	                    IF (#sx_Gapping_Rvs          // Gapping needs to be applied bit
	                        AND ((#sdi_GapHeadToHeadConfiguration_Rvs > #sdi_GapHeadToHead_Rvs    // Configured head to head bigger than the actual one
	                        OR #sdi_GapHeadToHeadConfiguration_Rvs - #idi_PEC_BoSDistance / 10 + #sdi_PECtoEndDistance_Rvs > #sdi_DownstreamGapHeadToHead_Rvs
	                        OR #sdi_GapTailToHeadConfiguration_Rvs > #sdi_Gap_Rvs     // Configured gap bigger than the actual one
	                        OR #sdi_GapTailToHeadConfiguration_Rvs - #idi_PEC_BoSDistance / 10 + #sdi_PECtoEndDistance_Rvs > #sdi_DownstreamGapTailtoHead_Rvs)
	                        AND NOT #sx_RecoveryGap_Rvs)                                                // Die back recovery gap bit not active
	                        OR (((#sdi_GapHeadToHeadConfiguration_Rvs + #i_UDT_ConveyorConfiguration.ExtraGapRecovery)   // Add recovery gap to the configured
	                        > #sdi_GapHeadToHead_Rvs                                                                                 // Actual head to head distance
	                        OR (#sdi_GapHeadToHeadConfiguration_Rvs - #idi_PEC_BoSDistance / 10 + #sdi_PECtoEndDistance_Rvs + #i_UDT_ConveyorConfiguration.ExtraGapRecovery)
	                        > #sdi_DownstreamGapHeadToHead_Rvs
	                        OR (#sdi_GapTailToHeadConfiguration_Rvs + #i_UDT_ConveyorConfiguration.ExtraGapRecovery)    // Add recovery gap to the configured
	                        > #sdi_Gap_Rvs                                                                               // Actual gap between parcels
	                        OR (#sdi_GapTailToHeadConfiguration_Rvs - #idi_PEC_BoSDistance / 10 + #sdi_PECtoEndDistance_Rvs + #i_UDT_ConveyorConfiguration.ExtraGapRecovery)
	                        > #sdi_DownstreamGapTailtoHead_Rvs)
	                        AND #sx_RecoveryGap_Rvs))                                                                                // Recovery gap bit activate
	                    THEN

	                        #sdi_GapHeadToHead_Rvs -= #iq_UDT_HandShakeUp.DownstreamDisplacement;      // Increase head to head counter with conveyor downstream displacement
	                        #sdi_Gap_Rvs -= #iq_UDT_HandShakeUp.DownstreamDisplacement;     // Increase gap counter with conveyor downstream displacement

	                    ELSE

	                        #sx_Gapping_Rvs := FALSE;                   // Set gapping bit to false

	                    END_IF;

	                    IF #sx_Gapping_Rvs                              // Gapping bit active
	                        AND NOT #iq_UDT_HandShakeUp.RTR           // Ready to receive not active
	                    THEN

	                        #sx_RecoveryGap_Rvs := TRUE;                // Recovery gap activation after die back

	                    END_IF;

	                    IF #sx_RecoveryGap_Rvs                          // Recovery gap active
	                        AND NOT #sx_Gapping_Rvs                     // Gapping bit not active
	                    THEN

	                        #sx_RecoveryGap_Rvs := FALSE;               // Recovery gap disable

	                    END_IF;

	                END_REGION
	            END_IF;
	        END_REGION

	        REGION 7.6 - Ready to send and Transfer in progress
	            IF NOT #sx_ReverseDirection
	            THEN
	                REGION 7.6.1 - Forward

	                    IF #iq_UDT_HandShake.RTR                                            // Ready to receive bit
	                        AND NOT #sx_Gapping_Fwd
	                        AND #sx_AuxHeadAtEnd_Fwd                                            // Parcel is at end of conveyor
	                        AND NOT #ix_ExternalRequestDieBack
	                    THEN

	                        #iq_UDT_HandShake.TIP := TRUE;      // Transfer in progress bit
	                        #iq_UDT_HandShake.RTS := FALSE;     // Ready to send bit
	                        #sx_AuxHeadAtEnd_Fwd := FALSE;

	                    END_IF;

	                    IF #R_TRIG_TailToBegin_Fwd.Q               // Reset TIP when the parcel leaves interlock
	                    THEN

	                        #iq_UDT_HandShake.TIP := FALSE;     // Transfer in progress bit

	                    END_IF;

	                END_REGION
	            ELSE
	                REGION 7.6.2 - Reverse

	                    IF #iq_UDT_HandShakeUp.RTR                                            // Ready to receive bit
	                        AND #iq_UDT_HandShake.RTR
	                        AND NOT #sx_Gapping_Rvs
	                        AND #sx_AuxHeadAtEnd_Rvs                                            // Parcel is at end of conveyor
	                        AND NOT #ix_ExternalRequestDieBack
	                    THEN

	                        #iq_UDT_HandShakeUp.TIP := TRUE;      // Transfer in progress bit
	                        #iq_UDT_HandShakeUp.RTS := FALSE;     // Ready to send bit
	                        #sx_AuxHeadAtEnd_Rvs := FALSE;

	                    END_IF;

	                    IF #R_TRIG_TailToBegin_Rvs.Q               // Reset TIP when the parcel leaves interlock
	                    THEN

	                        #iq_UDT_HandShakeUp.TIP := FALSE;     // Transfer in progress bit

	                    END_IF;

	                END_REGION
	            END_IF;
	        END_REGION

	        REGION 7.7 - Downstream gap

	            (* This functionality is used to maintain the gap between parcel conveyor's downstream.
	               To do this, is used the downstream displacement.  *)
	            IF NOT #sx_ReverseDirection
	            THEN
	                REGION 7.7.1 - Forward

	                    IF #R_TRIG_TailToBegin_Fwd.Q                       // When the parcel's tail reach the beginning of downstream conveyor
	                    THEN

	                        #sdi_DownstreamGapTailtoHead_Fwd := 0;                     // Reset downstream gap counter

	                    END_IF;

	                    IF #sdi_DownstreamGapTailtoHead_Fwd < #ci_OverflowLimit        // Prevent integer variable overflow
	                    THEN

	                        #sdi_DownstreamGapTailtoHead_Fwd += #iq_UDT_HandShake.DownstreamDisplacement;          // Downstream displacement gap counter

	                    END_IF;

	                END_REGION
	            ELSE
	                REGION 7.7.2 - Reverse

	                    IF #R_TRIG_TailToBegin_Rvs.Q                       // When the parcel's tail reach the beginning of downstream conveyor
	                    THEN

	                        #sdi_DownstreamGapTailtoHead_Rvs := 0;                     // Reset downstream gap counter

	                    END_IF;

	                    IF #sdi_DownstreamGapTailtoHead_Rvs < #ci_OverflowLimit        // Prevent integer variable overflow
	                    THEN

	                        #sdi_DownstreamGapTailtoHead_Rvs -= #iq_UDT_HandShakeUp.DownstreamDisplacement;          // Downstream displacement gap counter

	                    END_IF;

	                END_REGION
	            END_IF;
	        END_REGION

	        REGION 7.8 - Downstream Head to Head
	            IF NOT #sx_ReverseDirection
	            THEN
	                REGION 7.8.1 - Forward

	                    #R_TRIG_Transfering_Fwd(CLK := #iq_UDT_HandShake.TIP);

	                    IF #R_TRIG_Transfering_Fwd.Q                                                           // Transfering aux bit rising trigger
	                    THEN

	                        #sdi_DownstreamGapHeadToHead_Fwd := 0;                                              // Downstream head to head reset counter

	                    END_IF;

	                    IF #sdi_DownstreamGapHeadToHead_Fwd < #ci_OverflowLimit                                 // Prevent integer variable overflow
	                    THEN

	                        #sdi_DownstreamGapHeadToHead_Fwd += #iq_UDT_HandShake.DownstreamDisplacement;       // Downstream displacement head to head counter

	                    END_IF;

	                END_REGION
	            ELSE
	                REGION 7.8.2 - Reverse

	                    #R_TRIG_Transfering_Rvs(CLK := #iq_UDT_HandShake.TIP);

	                    IF #R_TRIG_Transfering_Rvs.Q                                                           // Transfering aux bit rising trigger
	                    THEN

	                        #sdi_DownstreamGapHeadToHead_Rvs := 0;                                              // Downstream head to head reset counter

	                    END_IF;

	                    IF #sdi_DownstreamGapHeadToHead_Rvs < #ci_OverflowLimit                                 // Prevent integer variable overflow
	                    THEN

	                        #sdi_DownstreamGapHeadToHead_Rvs -= #iq_UDT_HandShakeUp.DownstreamDisplacement;       // Downstream displacement head to head counter

	                    END_IF;

	                END_REGION
	            END_IF;
	        END_REGION

	        REGION 7.9 - Energy save

	            (* Save energy functionality is used to stop conveyor if no parcels are in the system to save energy
	               Save energy function counts displacement if the photo eye do not detects parcels. The counter is reset if:
	               - Photo eye is triggered.
	               - Reset is required from external.
	               - Ready to send is active from upstream. *)

	            // Energy save sensors filter
	            IF NOT #ix_PEC_EoS OR NOT #ix_PEC_BoS
	            THEN
	                #si_EnergySaveFilter += ABS(IN := #iq_UDT_ConveyorInterface.Displacement);
	            ELSE
	                #si_EnergySaveFilter := 0;
	            END_IF;

	            IF #i_UDT_ConveyorConfiguration.Energy                                       // Energy save functionality enable from configuration
	            THEN

	                IF #sdi_AuxEnergySave_Fwd >= #i_UDT_ConveyorConfiguration.Forward_Direction.EnergySaveLenght        // Compare energy save counter with configured lenght
	                    OR #sdi_AuxEnergySave_Rvs >= #i_UDT_ConveyorConfiguration.Reverse_Direction.EnergySaveLenght
	                THEN
	                    #sx_EnergySaveActive := TRUE;                                           // Set energy save active true
	                END_IF;

	                IF ((#si_EnergySaveFilter >= #ci_MinimumParcelLength)                                  // Photo eye detects a parcel
	                    AND NOT #sx_EnergySaveActive)                                         // Energy save active bit
	                    OR #ix_ResetEnergySave                                               // Reset energy save
	                    OR (#iq_UDT_HandShakeUp.ResetEnergySave AND NOT #sx_ReverseDirection)                               // Reset energy save externaly
	                    OR (#iq_UDT_HandShake.ResetEnergySave AND #sx_ReverseDirection)
	                    OR NOT #iq_UDT_EquipmentControl.Command.AutomaticOn                  // Automatic ON from control block
	                    OR #iq_UDT_EquipmentControl.Command.Stop                             // Stop command from control block
	                THEN
	                    #sdi_AuxEnergySave_Fwd := 0;                                        // Reset energy save counter
	                    #sdi_AuxEnergySave_Rvs := 0;                                        // Reset energy save counter
	                    #sx_EnergySaveActive := FALSE;                                      // Set energy save active to false
	                ELSE
	                    // Increament displacement counter
	                    IF NOT #sx_ReverseDirection
	                    THEN
	                        #sdi_AuxEnergySave_Fwd += #iq_UDT_ConveyorInterface.Displacement;
	                    ELSE
	                        #sdi_AuxEnergySave_Rvs -= #iq_UDT_ConveyorInterface.Displacement;
	                    END_IF;
	                END_IF;

	            ELSE
	                // If energy save functionality is disable from configuration
	                #sdi_AuxEnergySave_Fwd := 0;
	                #sdi_AuxEnergySave_Rvs := 0;// Reset energy save counter
	                #sx_EnergySaveActive := FALSE;                                      // Set energy save false
	            END_IF;
	            // Reset to downstream when not already in enery save on signal of PEC
	            // When slave conveyor pass reset esave command to master conveyor

	            IF NOT #sx_ReverseDirection
	            THEN
	                #iq_UDT_HandShake.ResetEnergySave := (NOT #ix_PEC_EoS OR #sx_AuxHeadAtEnd_Fwd OR #iq_UDT_HandShake.TIP) AND NOT #sx_EnergySaveActive
	                OR (#i_UDT_ConveyorConfiguration.Forward_Direction.Mode = 1 AND #iq_UDT_HandShakeUp.ResetEnergySave);
	            ELSE
	                #iq_UDT_HandShakeUp.ResetEnergySave := (NOT #ix_PEC_BoS OR #sx_AuxHeadAtEnd_Rvs OR #iq_UDT_HandShakeUp.TIP) AND NOT #sx_EnergySaveActive
	                OR (#i_UDT_ConveyorConfiguration.Reverse_Direction.Mode = 1 AND #iq_UDT_HandShake.ResetEnergySave);
	            END_IF;
	        END_REGION

	        REGION 7.10 - Operation modes

	            // Different modes in automatic can be configured
	            // 1 - Slave
	            // 2 - Queue
	            // 3 - Bulk flow

	            IF #sx_AutomaticActive                                          // Automatic mode active
	                AND #tx_CascadeStart                                        // Cascade startup
	            THEN

	                IF NOT #sx_ReverseDirection
	                THEN

	                    CASE #i_UDT_ConveyorConfiguration.Forward_Direction.Mode OF                   // Operation mode configured

	                        1:  // Slave

	                            // Run conveyor if ready to receive if on, and conveyor is not gapping,
	                            // and not halt request and not energy save active

	                            #iq_UDT_ConveyorInterface.RunFwd := #sx_AutomaticActive     // Automatic mode active
	                            AND #sx_Ready                                               // Ready active
	                            AND NOT #ix_ExternalRequestHold                             // Halt request is not active
	                            AND NOT #sx_EnergySaveActive                                // Energy save not active
	                            AND #iq_UDT_HandShake.RTR                               // Ready to receive active
	                            AND NOT #sx_DirectionChanged;

	                            #iq_UDT_HandShakeUp.RTR := #iq_UDT_ConveyorInterface.RunFwd;

	                        2:  // Master

	                            // With queue configuration, conveyor runs if ready to receive is true.
	                            // If ready to receive is false, conveyor runs until parcel reach the end of the conveyor.

	                            // Conveyor stops if heads parcel reache the end of the conveyor and:
	                            // - Ready to receive is false
	                            // - Or die back requested.
	                            // - Or halt requested
	                            // Conveyor also stops if gapping is active or energy save mode active.

	                            #iq_UDT_ConveyorInterface.RunFwd := #sx_AutomaticActive             // Automatic mode active
	                            AND #sx_Ready                                                       // Ready active
	                            AND NOT #sx_DirectionChanged
	                            AND NOT #sx_Gapping_Fwd                                                 // Gapping request
	                            AND NOT #sx_EnergySaveActive                                        // Energy save request
	                            AND NOT #ix_ExternalRequestHold                                     // Halt requested from external
	                            AND ((NOT #ix_ExternalRequestDieBack
	                            AND #iq_UDT_HandShake.RTR)
	                            OR (NOT #sx_AuxHeadAtEnd_Fwd
	                            AND NOT #iq_UDT_HandShake.TIP)
	                            OR (#iq_UDT_HandShake.RTR
	                            AND NOT #sx_AuxHeadAtEnd_Fwd));

	                            #iq_UDT_HandShakeUp.RTR := #iq_UDT_ConveyorInterface.RunFwd;


	                        3: //Master at bulk flow

	                            #iq_UDT_ConveyorInterface.RunFwd := #sx_AutomaticActive             // Automatic mode active
	                            AND #sx_Ready                                                       // Ready active
	                            AND NOT #sx_DirectionChanged
	                            AND NOT #sx_EnergySaveActive                                        // Energy save request
	                            AND NOT #ix_ExternalRequestHold                                     // Halt requested from external
	                            AND (
	                            (NOT #ix_ExternalRequestDieBack                                     //no die back request and the downstream is running
	                            AND #iq_UDT_HandShake.RTR)
	                            OR                                                                  //..or..
	                            (#sdi_TransitionZone = 0)                                            // no parcels at the transition zone
	                            OR                                                                  //..or..
	                            (#iq_UDT_HandShake.RTR
	                            AND NOT #ix_ExternalRequestDieBack
	                            AND NOT (#sdi_TransitionZone = 0)));                                  //downstream is running and there are

	                            //If PEC is blocked, reset tracking counter
	                            IF NOT #ix_PEC_EoS THEN
	                                #sdi_TransitionZone := #sdi_PEC_EoSDistance_Fwd / 10;
	                            END_IF;

	                            //Track parcels at the zone between EoS and conveyor end (Transition Zone)
	                            #sdi_TransitionZone := #sdi_TransitionZone - ABS(#iq_UDT_ConveyorInterface.Displacement);

	                            //If Value is negative then set to 0
	                            IF #sdi_TransitionZone < 0 THEN
	                                #sdi_TransitionZone := 0;
	                            END_IF;

	                            #iq_UDT_HandShakeUp.RTR := #iq_UDT_ConveyorInterface.RunFwd;

	                    END_CASE;

	                ELSE

	                    CASE #i_UDT_ConveyorConfiguration.Reverse_Direction.Mode OF                   // Operation mode configured

	                        1:  // Slave

	                            // Run conveyor if ready to receive if on, and conveyor is not gapping,
	                            // and not halt request and not energy save active

	                            #iq_UDT_ConveyorInterface.RunRvs := #sx_AutomaticActive     // Automatic mode active
	                            AND #sx_Ready                                               // Ready active
	                            AND NOT #ix_ExternalRequestHold                             // Halt request is not active
	                            AND NOT #sx_EnergySaveActive                                // Energy save not active
	                            AND #iq_UDT_HandShakeUp.RTR                                 // Ready to receive active
	                            AND NOT #sx_DirectionChanged;

	                            #iq_UDT_HandShake.RTR := #iq_UDT_ConveyorInterface.RunRvs;

	                        2:  // Master

	                            // With queue configuration, conveyor runs if ready to receive is true.
	                            // If ready to receive is false, conveyor runs until parcel reach the end of the conveyor.

	                            // Conveyor stops if heads parcel reache the end of the conveyor and:
	                            // - Ready to receive is false
	                            // - Or die back requested.
	                            // - Or halt requested
	                            // Conveyor also stops if gapping is active or energy save mode active.

	                            #iq_UDT_ConveyorInterface.RunRvs := #sx_AutomaticActive             // Automatic mode active
	                            AND #sx_Ready                                                       // Ready active
	                            AND NOT #sx_DirectionChanged
	                            AND NOT #sx_Gapping_Rvs                                             // Gapping request
	                            AND NOT #sx_EnergySaveActive                                        // Energy save request
	                            AND NOT #ix_ExternalRequestHold                                     // Halt requested from external
	                            AND ((NOT #ix_ExternalRequestDieBack
	                            AND #iq_UDT_HandShakeUp.RTR)
	                            OR (NOT #sx_AuxHeadAtEnd_Rvs
	                            AND NOT #iq_UDT_HandShakeUp.TIP)
	                            OR (#iq_UDT_HandShakeUp.RTR
	                            AND NOT #sx_AuxHeadAtEnd_Rvs));

	                            #iq_UDT_HandShake.RTR := #iq_UDT_ConveyorInterface.RunRvs;


	                        3: //Master at bulk flow

	                            #iq_UDT_ConveyorInterface.RunRvs := #sx_AutomaticActive             // Automatic mode active
	                            AND #sx_Ready                                                       // Ready active
	                            AND NOT #sx_DirectionChanged
	                            AND NOT #sx_EnergySaveActive                                        // Energy save request
	                            AND NOT #ix_ExternalRequestHold                                     // Halt requested from external
	                            AND (
	                            (NOT #ix_ExternalRequestDieBack                                     //no die back request and the downstream is running
	                            AND #iq_UDT_HandShakeUp.RTR)
	                            OR                                                                  //..or..
	                            (#sdi_TransitionZone = 0)                                            // no parcels at the transition zone
	                            OR                                                                  //..or..
	                            (#iq_UDT_HandShakeUp.RTR
	                            AND NOT #ix_ExternalRequestDieBack
	                            AND NOT (#sdi_TransitionZone = 0)));                                  //downstream is running and there are

	                            //If PEC is blocked, reset tracking counter
	                            IF NOT #ix_PEC_BoS THEN
	                                #sdi_TransitionZone := #sdi_PEC_EoSDistance_Rvs / 10;
	                            END_IF;
	                            //Track parcels at the zone between EoS and conveyor end (Transition Zone)
	                            #sdi_TransitionZone := #sdi_TransitionZone - ABS(#iq_UDT_ConveyorInterface.Displacement);

	                            //If Value is negative then set to 0
	                            IF #sdi_TransitionZone < 0 THEN
	                                #sdi_TransitionZone := 0;
	                            END_IF;

	                            #iq_UDT_HandShake.RTR := #iq_UDT_ConveyorInterface.RunRvs;
	                    END_CASE;

	                END_IF;

	            ELSE

	                // If conveyor is not in manual mode and not ready
	                IF NOT #sx_ReverseDirection
	                THEN
	                    #iq_UDT_ConveyorInterface.RunFwd := FALSE;                      // Order to VFD stop conveyor
	                    #iq_UDT_HandShakeUp.RTR := FALSE;                               // Set ready to receive false
	                ELSE
	                    #iq_UDT_ConveyorInterface.RunRvs := FALSE;                      // Order to VFD stop conveyor
	                    #iq_UDT_HandShake.RTR := FALSE;                               // Set ready to receive false
	                END_IF;

	            END_IF;

	        END_REGION

	    END_IF;
	END_REGION

	REGION 8 - Speed control

	    (*In manual mode, conveyor default runs with manual speed which is calculated as a percentage of nominal speed. If "ManualFullSpeed" is set true, conveyor runs with high speed in manual mode.
	     In jog mode conveyor always runs in low speed. In automatic mode, conveyor runs with full speed if external is zero. If external speed is bigger than zero, conveyor will run with that speed. *)


	    // security
	    IF #iq_UDT_ConveyorCommand.ManualSpeed > 100 THEN
	        #iq_UDT_ConveyorCommand.ManualSpeed := 100;
	    END_IF;

	    IF #iq_UDT_ConveyorCommand.ManualSpeed < 0 THEN
	        #iq_UDT_ConveyorCommand.ManualSpeed := 0;
	    END_IF;



	    IF #sx_ManualModeActive                                                                         // Manual mode active
	    THEN

	        IF #iq_UDT_ConveyorCommand.ManualStartStop                                              // Full speed in manual mode
	        THEN

	            IF #iq_UDT_ConveyorCommand.ManualFullSpeed                                                  // Full speed in manual mode
	            THEN
	                #iq_UDT_ConveyorInterface.SpeedSetpoint := #i_UDT_ConveyorConfiguration.SpeedSetpointNominal;    // Move nominal setpoint to the VDF

	            ELSE
	                #iq_UDT_ConveyorInterface.SpeedSetpoint := REAL_TO_INT(INT_TO_REAL(#iq_UDT_ConveyorCommand.ManualSpeed) * (INT_TO_REAL(#i_UDT_ConveyorConfiguration.SpeedSetpointNominal) / 100));     // Calculate and Move manual speed setpoint to VFD

	            END_IF;

	        ELSE                                                                                             //low speed for jog mode

	            IF #i_UDT_ConveyorConfiguration.SpeedSetpointLow < #i_UDT_ConveyorConfiguration.SpeedSetpointNominal  //Low speed can't be higher than nominal speed
	            THEN
	                #iq_UDT_ConveyorInterface.SpeedSetpoint := #i_UDT_ConveyorConfiguration.SpeedSetpointLow;    // Move low speed setpoint to the VDF

	            ELSE

	                #iq_UDT_ConveyorInterface.SpeedSetpoint := #i_UDT_ConveyorConfiguration.SpeedSetpointNominal;    // Move low speed setpoint to the VDF
	            END_IF;
	        END_IF;



	    ELSE

	        IF #ii_ExternalSpeed > 0                                                                      // If external speed bigger than zero
	        THEN
	            #iq_UDT_ConveyorInterface.SpeedSetpoint := #ii_ExternalSpeed;                                     // Move external speed to VFD
	        ELSE
	            #iq_UDT_ConveyorInterface.SpeedSetpoint := #i_UDT_ConveyorConfiguration.SpeedSetpointNominal;       // Move nominal setpoint to VFD
	        END_IF;

	    END_IF;



	END_REGION


	REGION 9 - Status
	    #s_UDT_HMIStatus.Specific.Reverse := #sx_ReverseDirection;

	    // stopped
	    #s_UDT_CommonStatus.Stopped := NOT #sx_Ready OR NOT #sx_AutomaticActive;

	    // Auto ON
	    #s_UDT_CommonStatus.AutoON := #sx_Ready AND #sx_AutomaticActive;

	    // Running
	    #s_UDT_CommonStatus.Running := #iq_UDT_ConveyorInterface.RunFwd
	    OR #iq_UDT_ConveyorInterface.RunRvs;

	    // Halted
	    #s_UDT_CommonStatus.Halted := #ix_ExternalRequestHold
	    AND #s_UDT_CommonStatus.AutoON
	    AND NOT #s_UDT_CommonStatus.EnergySave;

	    // Energy save active
	    #s_UDT_CommonStatus.EnergySave := #sx_EnergySaveActive AND #sx_AutomaticActive;

	    // Die back
	    #s_UDT_CommonStatus.Dieback := #s_UDT_CommonStatus.AutoON
	    AND NOT #s_UDT_CommonStatus.EnergySave
	    AND NOT #s_UDT_CommonStatus.Running;

	    // Manual
	    #s_UDT_CommonStatus.Manual := #sx_ManualModeActive;

	    // Manual Running
	    #s_UDT_CommonStatus.ManualRun := #sx_ManualModeActive AND #s_UDT_CommonStatus.Running;

	    // Safety not ok
	    #s_UDT_CommonStatus.SafetyStop := NOT #ix_SafetyOk AND #ix_HardwareOk;

	    // HMI status update
	    IF #s_UDT_CommonStatusOld <> #s_UDT_CommonStatus                                            // update on change
	        OR (#R_TRIG_Reverse.Q OR #F_TRIG_Reverse.Q)
	    THEN
	        // HMI status initialization
	        #s_UDT_HMIStatus.Status := 0;


	        // Energy save
	        IF #s_UDT_CommonStatus.EnergySave
	        THEN
	            #s_UDT_HMIStatus.Status := "DB_HMIStatusConfiguration".EnergySave;
	        END_IF;

	        // Running
	        IF #s_UDT_CommonStatus.Running
	        THEN
	            #s_UDT_HMIStatus.Status := "DB_HMIStatusConfiguration".Running;
	        END_IF;

	        // Stopped
	        IF #s_UDT_CommonStatus.Stopped
	        THEN
	            #s_UDT_HMIStatus.Status := "DB_HMIStatusConfiguration".Stopped;
	        END_IF;

	        // Dieback
	        IF #s_UDT_CommonStatus.Dieback
	        THEN
	            #s_UDT_HMIStatus.Status := "DB_HMIStatusConfiguration".Dieback;
	        END_IF;

	        // Halted
	        IF #s_UDT_CommonStatus.Halted
	        THEN
	            #s_UDT_HMIStatus.Status := "DB_HMIStatusConfiguration".Halted;
	        END_IF;

	        // Manual
	        IF #s_UDT_CommonStatus.Manual
	        THEN
	            #s_UDT_HMIStatus.Status := "DB_HMIStatusConfiguration".Manual;
	        END_IF;

	        // Running in manual mode
	        IF #s_UDT_CommonStatus.ManualRun
	        THEN
	            #s_UDT_HMIStatus.Status := "DB_HMIStatusConfiguration".ManualRun;
	        END_IF;

	(*        // Internal tracking warning
	        IF #iq_UDT_ConveyorInterface.InternalWarningTracking
	        THEN
	            #s_UDT_HMIStatus.Status := "DB_HMIStatusConfiguration".Warning;
	        END_IF; *)

	        // Internal tracking error
	        IF #iq_UDT_ConveyorInterface.InternalErrorTracking
	        THEN
	            #s_UDT_HMIStatus.Status := "DB_HMIStatusConfiguration".TrackingError;
	        END_IF;

	        // Internal PEC error
	        IF #iq_UDT_ConveyorInterface.InternalErrorPEC
	        THEN
	            #s_UDT_HMIStatus.Status := "DB_HMIStatusConfiguration".PECJam;
	        END_IF;

	        // Internal Encoder error
	        IF #iq_UDT_ConveyorInterface.InternalErrorEncoder
	        THEN
	            #s_UDT_HMIStatus.Status := "DB_HMIStatusConfiguration".EncoderError;
	        END_IF;

	        // Internal VFD error
	        IF #iq_UDT_ConveyorInterface.InternalErrorVFD
	        THEN
	            #s_UDT_HMIStatus.Status := "DB_HMIStatusConfiguration".VFDError;
	        END_IF;

	        // Disconnect error
	        IF #iq_UDT_ConveyorInterface.Disconnected
	        THEN
	            #s_UDT_HMIStatus.Status := "DB_HMIStatusConfiguration".CBError;
	        END_IF;

	        // Safety stop
	        IF (#s_UDT_CommonStatus.SafetyStop)
	        THEN
	            #s_UDT_HMIStatus.Status := "DB_HMIStatusConfiguration".SafetyStop;
	        END_IF;

	        #s_UDT_CommonStatusOld := #s_UDT_CommonStatus;              // Copy status to memory
	        #q_UDT_Status := #s_UDT_CommonStatus;                       // Copy status to output

	    END_IF;

	    // Copy HMI status to output
	    #q_UDT_HMIStatus := #s_UDT_HMIStatus;

	END_REGION


	REGION 10 - Statistics

	    REGION 10.1 - Conveyor up time

	        IF #sx_Up OR #iq_UDT_EquipmentControl.Command.ResetData    // Reset statistics
	        THEN

	            "FC_Statistics"(ix_Reset := #iq_UDT_EquipmentControl.Command.ResetData,      // Reset statistics input
	                            ix_Activate := #sx_Up,
	                            ix_RTrigActivate := #R_TRIG_ConveyorUp.Q,                     // Statistics active trigger
	                            iqUDT_Statistics := #iq_UDT_Statistics.ConveyorUp);      // Statistics values output

	        END_IF;

	    END_REGION

	    REGION 10.2 - Energy save

	        // Statistics Energy save mode active
	        IF #s_UDT_CommonStatus.EnergySave(* #sx_EnergySaveActive *)                                                        // Energy save active
	            OR #iq_UDT_EquipmentControl.Command.ResetData                               // Reset statistics
	        THEN
	            "FC_Statistics"(ix_Reset := #iq_UDT_EquipmentControl.Command.ResetData,      // Reset statistics input
	                            ix_Activate := #s_UDT_CommonStatus.EnergySave,                         // Activate statistics functions input
	                            ix_RTrigActivate := #R_TRIG_EnergySave.Q,                    // Statistics active trigger
	                            iqUDT_Statistics := #iq_UDT_Statistics.EnergySave);         // Statistics values output

	        END_IF;

	    END_REGION

	    REGION 10.3 - Conveyor down time

	        // Conveyor down is when conveyor is not in manual mode and has an error
	        IF #sx_Down OR #iq_UDT_EquipmentControl.Command.ResetData OR #s_UDT_CommonStatus.SafetyStop                                    // Reset statistics
	        THEN

	            "FC_Statistics"(ix_Reset := #iq_UDT_EquipmentControl.Command.ResetData,             // Reset statistics input
	                            ix_Activate := #sx_Down OR #s_UDT_CommonStatus.SafetyStop, // Activate statistics functions input
	                            ix_RTrigActivate := #R_TRIG_ConveyorDownTime.Q,                     // Statistics active trigger
	                            iqUDT_Statistics := #iq_UDT_Statistics.ConveyorDown);              // Statistics values output

	        END_IF;
	    END_REGION

	    REGION 10.4 - Conveyor stop time

	        IF #sx_Stopped OR #iq_UDT_EquipmentControl.Command.ResetData                                           // Reset statistics
	        THEN

	            "FC_Statistics"(ix_Reset := #iq_UDT_EquipmentControl.Command.ResetData,        // Reset statistics input
	                            ix_Activate := #sx_Stopped,                                           // Activate statistics functions input
	                            ix_RTrigActivate := #R_TRIG_ConveyorStopped.Q,                        // Statistics active trigger
	                            iqUDT_Statistics := #iq_UDT_Statistics.ConveyorStop);                  // Statistics values output

	        END_IF;
	    END_REGION

	END_REGION

	REGION 11 - Report to control block
	    // Function to manage report between control block and conveyor block
	    "FC_EquipmentReport"(iUDT_Status := #s_UDT_CommonStatus,
	                         iqUDT_Control := #iq_UDT_EquipmentControl);

	END_REGION

	REGION 12 - Internal errors and warnings reset

	    IF #iq_UDT_EquipmentControl.Command.Reset
	    THEN

	        #iq_UDT_ConveyorInterface.InternalErrorEncoder := FALSE;
	        #iq_UDT_ConveyorInterface.InternalErrorPEC := FALSE;
	        #iq_UDT_ConveyorInterface.InternalWarningTracking := FALSE;
	        #iq_UDT_ConveyorInterface.InternalErrorTracking := FALSE;
	        #iq_UDT_ConveyorInterface.InternalWarningVFD := FALSE;
	        #iq_UDT_ConveyorInterface.InternalErrorVFD := FALSE;
	        #iq_UDT_ConveyorInterface.Disconnected := FALSE;
	        #iq_UDT_ConveyorInterface.ConfigurationError := FALSE;
	    END_IF;

	END_REGION






END_FUNCTION_BLOCK

FUNCTION_BLOCK "FB_ConnectionCheck1Hz"
{ S7_Optimized_Access := 'TRUE' }
VERSION : 3.2
// ATTRIBUTES
// AUTO_NUMBER = True
// BLOCK_NUMBER = 93
// END_ATTRIBUTES
   VAR_INPUT
      ix_LifebitIn { ExternalAccessible := 'False'; ExternalVisible := 'False'; ExternalWritable := 'False'} : Bool;   // Input life bit
      ix_IOModuleOK { ExternalAccessible := 'False'; ExternalVisible := 'False'; ExternalWritable := 'False'} : Bool;   // TRUE when IO module is Ok
   END_VAR

   VAR_OUTPUT
      qx_LifebitOut { ExternalAccessible := 'False'; ExternalVisible := 'False'; ExternalWritable := 'False'} : Bool;   // Generated life bit 1 sec ON/1 sec OFF
   END_VAR

   VAR_IN_OUT
      iqudt_ConnectionStatus : "UDT_ConnectStatus";   // Connection status
   END_VAR

   VAR
      FB_Pulse_Instance { ExternalAccessible := 'False'; ExternalVisible := 'False'; ExternalWritable := 'False'; S7_SetPoint := 'False'} : "FB_Pulse";
      F_TRIG_LifebitIn {InstructionName := 'F_TRIG'; LibVersion := '1.0'; ExternalAccessible := 'False'; ExternalVisible := 'False'; ExternalWritable := 'False'; S7_SetPoint := 'False'} : F_TRIG;   // Falling edge trigger Lifebit in
      R_TRIG_LifebitIn {InstructionName := 'R_TRIG'; LibVersion := '1.0'; ExternalAccessible := 'False'; ExternalVisible := 'False'; ExternalWritable := 'False'; S7_SetPoint := 'False'} : R_TRIG;   // Rising edge trigger  Lifebit in
      sx_LifebitValue { ExternalAccessible := 'False'; ExternalVisible := 'False'; ExternalWritable := 'False'} : Bool;   // Lifebit value
      sx_ConnectionFault { ExternalAccessible := 'False'; ExternalVisible := 'False'; ExternalWritable := 'False'} : Bool;   // Connection Fault
   END_VAR

   VAR_TEMP
      tx_Pulse : Bool;   // Generated pulse signal
   END_VAR

   VAR CONSTANT
      cudi_ConnectionFaultOnDelay : UDInt := 5000;   // Connection On Delay
   END_VAR


BEGIN
	(*
	----------------------------------------------------------------------------------------
	|                                                                                      |
	|  Copyright  2023             FORTNA Europe BV                                        |
	|  All Rights Reserved         Netherlands                                             |
	|                                                                                      |
	----------------------------------------------------------------------------------------

	Version history:
	Date        | Version   | Author        | Remark
	----------------------------------------------------------------------------------------
	12/10/2023  | 1.0       | S. Nikodem    | First release TIA 17 | DHL Munich
	12/03/2024  | 1.1       | S. Nieswiec      | Added to new Baseline
	*)

	REGION 1 - Life bit generations

	    //Generation
	    #qx_LifebitOut := "DB_Memory".Clock_1Hz;

	END_REGION

	REGION 2 - Hardware Ok

	    IF NOT #ix_IOModuleOK THEN

	        //Status update
	        #iqudt_ConnectionStatus.Specific.CommunicationFault := False;
	        #iqudt_ConnectionStatus.Specific.Connected := False;

	        #iqudt_ConnectionStatus.Status := 0;

	        RETURN;

	    END_IF;

	END_REGION

	REGION 3 - Connection check

	    //Trigger
	    #F_TRIG_LifebitIn(CLK := #ix_LifebitIn);
	    #R_TRIG_LifebitIn(CLK := #ix_LifebitIn);

	    IF (#F_TRIG_LifebitIn.Q OR #R_TRIG_LifebitIn.Q) THEN

	        #sx_LifebitValue := TRUE;
	    END_IF;

	    #FB_Pulse_Instance(iudi_PulseTime := #cudi_ConnectionFaultOnDelay,
	                       qx_Pulse => #tx_Pulse);

	    IF #tx_Pulse THEN
	        IF #sx_LifebitValue THEN

	            #sx_LifebitValue := False;

	            #sx_ConnectionFault := False;

	        ELSE

	            #sx_ConnectionFault := TRUE;

	        END_IF;
	    END_IF;

	END_REGION

	REGION 4 - Status update

	    #iqudt_ConnectionStatus.Specific.CommunicationFault := #sx_ConnectionFault;
	    #iqudt_ConnectionStatus.Specific.Connected := NOT #sx_ConnectionFault;

	    IF #sx_ConnectionFault
	    THEN
	        #iqudt_ConnectionStatus.Status := "DB_HMIStatusConfiguration".CommunicationError;
	    END_IF;

	    IF NOT #sx_ConnectionFault
	    THEN
	        #iqudt_ConnectionStatus.Status := "DB_HMIStatusConfiguration".AutoON;
	    END_IF;

	END_REGION
END_FUNCTION_BLOCK

FUNCTION_BLOCK "FB_Xray_Rapiscan"
{ S7_Optimized_Access := 'TRUE' }
VERSION : 0.1
// ATTRIBUTES
// AUTO_NUMBER = True
// BLOCK_NUMBER = 110
// END_ATTRIBUTES
   VAR_INPUT
      i_UDT_XrayConfiguration { ExternalAccessible := 'False'; ExternalVisible := 'False'; ExternalWritable := 'False'} : "UDT_XrayRapiscanConfiguration";   // Xray configuration structure
      ix_XrayEnergised { ExternalAccessible := 'False'; ExternalVisible := 'False'; ExternalWritable := 'False'} : Bool;   // Xray input signal - Energised
      ix_XrayFault { ExternalAccessible := 'False'; ExternalVisible := 'False'; ExternalWritable := 'False'} : Bool;   // Xray input signal - Fault
      ix_XrayReadyReceive { ExternalAccessible := 'False'; ExternalVisible := 'False'; ExternalWritable := 'False'} : Bool;   // Xray input signal - Ready receive
      ix_XrayReadySend { ExternalAccessible := 'False'; ExternalVisible := 'False'; ExternalWritable := 'False'} : Bool;   // Xray input signal - Ready send
      ix_XrayConveyorRunFwd { ExternalAccessible := 'False'; ExternalVisible := 'False'; ExternalWritable := 'False'} : Bool;   // Xray input signal - Conveyor run Fwd
      ix_XrayConveyorRunRvs { ExternalAccessible := 'False'; ExternalVisible := 'False'; ExternalWritable := 'False'} : Bool;   // Xray input signal - Conveyor run Rvs
      ix_XrayBagScaning { ExternalAccessible := 'False'; ExternalVisible := 'False'; ExternalWritable := 'False'} : Bool;   // Xray input signal - Xray bag scaning
      ix_XrayEmergencyStop { ExternalAccessible := 'False'; ExternalVisible := 'False'; ExternalWritable := 'False'} : Bool;   // Xray input signal - Emergency Stop
      ix_SafetyOk { ExternalAccessible := 'False'; ExternalVisible := 'False'; ExternalWritable := 'False'} : Bool;   // TRUE when Safety Circuit is healthy
      ix_24vOk { ExternalAccessible := 'False'; ExternalVisible := 'False'; ExternalWritable := 'False'} : Bool;   // TRUE when 24VDC is healthy
      ix_400vOk { ExternalAccessible := 'False'; ExternalVisible := 'False'; ExternalWritable := 'False'} : Bool;   // TRUE when 400VAC is healthy
      ix_HardwareOk { ExternalAccessible := 'False'; ExternalVisible := 'False'; ExternalWritable := 'False'} : Bool;   // TRUE when  hardware is Ok
      ix_SafetyReset { ExternalAccessible := 'False'; ExternalVisible := 'False'; ExternalWritable := 'False'} : Bool;   // TRUE Safety reset command is active
      is_ActualTime { ExternalAccessible := 'False'; ExternalVisible := 'False'; ExternalWritable := 'False'} : String;   // Actual date and time in String
   END_VAR

   VAR_OUTPUT
      q_UDT_HMIStatus { ExternalAccessible := 'False'; ExternalVisible := 'False'; ExternalWritable := 'False'} : "UDT_RapiscanStatus";   // HMI status structure
      qx_BHS_RDY_SEND { ExternalAccessible := 'False'; ExternalVisible := 'False'; ExternalWritable := 'False'} : Bool;   // Xray output signal - Input conveyor is ready to pass a bag to the Xray
      qx_BHS_RDY_RCV { ExternalAccessible := 'False'; ExternalVisible := 'False'; ExternalWritable := 'False'} : Bool;   // Xray output signal - Output conveyor is ready to accept a bag from the Xray
      qx_DECISION_ACK { ExternalAccessible := 'False'; ExternalVisible := 'False'; ExternalWritable := 'False'} : Bool;   // Xray output signal - Decision confirmation (only for Xray local control)
      qx_TRANSPORT_ENABLE { ExternalAccessible := 'False'; ExternalVisible := 'False'; ExternalWritable := 'False'} : Bool;   // Xray output signal - Transport mode eneble
      qx_TRANSPORT_FWD { ExternalAccessible := 'False'; ExternalVisible := 'False'; ExternalWritable := 'False'} : Bool;   // Xray output signal - Run forward request
      qx_TRANSPORT_REV { ExternalAccessible := 'False'; ExternalVisible := 'False'; ExternalWritable := 'False'} : Bool;   // Xray output signal - Run reverse request
      qx_ESTOP_IN { ExternalAccessible := 'False'; ExternalVisible := 'False'; ExternalWritable := 'False'} : Bool;   // Xray output signal - Estop
      qx_EMERGENCY_STOP_RESET { ExternalAccessible := 'False'; ExternalVisible := 'False'; ExternalWritable := 'False'} : Bool;   // Xray output signal - Estop resert
   END_VAR

   VAR_IN_OUT
      iq_UDT_Statistics : "UDT_RapiscanStatistics";   // Statistics structure
      iq_UDT_EquipmentControl : "UDT_EquipmentControl";   // Equipment control stucture
      iq_UDT_XrayConveyorInterface : "UDT_ConveyorInterface";   // Xray conveyor interface structure
      iq_UDT_Handshake : "UDT_ConveyorHandshake";   // Downstream handshake structure
      iq_UDT_HandShakeUp : "UDT_ConveyorHandshake";   // Upstream handshake structure
      iq_UDT_MFCCommand : "UDT_XrayCommand";   // Xray command structure
      iqs_XrayConveyorTrackingData : Array[*] of Int;   // Xray conveyor tracking array
      iq_UDT_XrayInterface : "UDT_XrayInterface";   // Xray interface structure
   END_VAR

   VAR
      s_EstopReset { ExternalAccessible := 'False'; ExternalVisible := 'False'; ExternalWritable := 'False'; S7_SetPoint := 'False'} : "FB_TimerOnOffDelay";   // Estop reset puls
      s_BagScaningTime { ExternalAccessible := 'False'; ExternalVisible := 'False'; ExternalWritable := 'False'; S7_SetPoint := 'False'} : "FB_TimerOnOffDelay";   // Bag scaning time
      s_UDT_HMIStatus { ExternalAccessible := 'False'; ExternalVisible := 'False'; ExternalWritable := 'False'; S7_SetPoint := 'False'} : "UDT_RapiscanStatus";   // HMI status structure
      s_UDT_CommonStatusOld { ExternalAccessible := 'False'; ExternalVisible := 'False'; ExternalWritable := 'False'; S7_SetPoint := 'False'} : "UDT_CommonStatus";   // Common status structure
      s_UDT_CommonStatus { ExternalAccessible := 'False'; ExternalVisible := 'False'; ExternalWritable := 'False'; S7_SetPoint := 'False'} : "UDT_CommonStatus";   // Common status structure
      R_TRIG_TransportMode {InstructionName := 'R_TRIG'; LibVersion := '1.0'; ExternalAccessible := 'False'; ExternalVisible := 'False'; ExternalWritable := 'False'; S7_SetPoint := 'False'} : R_TRIG;   // Rising edge trigger of Xray transport mode signal
      R_TRIG_XrayBagScaning {InstructionName := 'R_TRIG'; LibVersion := '1.0'; ExternalAccessible := 'False'; ExternalVisible := 'False'; ExternalWritable := 'False'; S7_SetPoint := 'False'} : R_TRIG;   // Rising edge trigger of Xray b ag scaning signal
      F_TRIG_XrayBagScaning {InstructionName := 'F_TRIG'; LibVersion := '1.0'; ExternalAccessible := 'False'; ExternalVisible := 'False'; ExternalWritable := 'False'; S7_SetPoint := 'False'} : F_TRIG;   // Falling edge trigger of Xray b ag scaning signal
      R_TRIG_SystemReadyRcv {InstructionName := 'R_TRIG'; LibVersion := '1.0'; ExternalAccessible := 'False'; ExternalVisible := 'False'; ExternalWritable := 'False'; S7_SetPoint := 'False'} : R_TRIG;   // Rising edge trigger of System ready to receive signal
      F_TRIG_SystemReadyRcv {InstructionName := 'F_TRIG'; LibVersion := '1.0'; ExternalAccessible := 'False'; ExternalVisible := 'False'; ExternalWritable := 'False'; S7_SetPoint := 'False'} : F_TRIG;   // Falling edge trigger of System ready to receive signal
      F_TRIG_ConveyorRunRvs {InstructionName := 'F_TRIG'; LibVersion := '1.0'; ExternalAccessible := 'False'; ExternalVisible := 'False'; ExternalWritable := 'False'; S7_SetPoint := 'False'} : F_TRIG;   // Falling edge trigger of Conveyor runs reverse direction signal
      ss_Counter { ExternalAccessible := 'False'; ExternalVisible := 'False'; ExternalWritable := 'False'} : Struct   // Statistics counters
         BagIDMessageNotReceived { ExternalAccessible := 'False'; ExternalVisible := 'False'; ExternalWritable := 'False'} : UDInt;   // Bag ID Message not received on time
         TransportmodeOn { ExternalAccessible := 'False'; ExternalVisible := 'False'; ExternalWritable := 'False'} : UDInt;   // Transport mode on
         TransportmodeOff { ExternalAccessible := 'False'; ExternalVisible := 'False'; ExternalWritable := 'False'} : UDInt;   // Transport mode off
         BackBelt { ExternalAccessible := 'False'; ExternalVisible := 'False'; ExternalWritable := 'False'} : UDInt;   // Backbelt functionality active
      END_STRUCT;
      si_GIN { ExternalAccessible := 'False'; ExternalVisible := 'False'; ExternalWritable := 'False'} : Int;   // GIN number
      sx_StartReceived { ExternalAccessible := 'False'; ExternalVisible := 'False'; ExternalWritable := 'False'} : Bool;   // Start command received from system
      sx_Ready { ExternalAccessible := 'False'; ExternalVisible := 'False'; ExternalWritable := 'False'} : Bool;   // Ready to operate in Automatic mode
      sx_AutomaticOn { ExternalAccessible := 'False'; ExternalVisible := 'False'; ExternalWritable := 'False'} : Bool;   // Automatic mode active
      sx_TransportmodeOn { ExternalAccessible := 'False'; ExternalVisible := 'False'; ExternalWritable := 'False'} : Bool;   // Transport mode active
      sx_TransportRunFwd { ExternalAccessible := 'False'; ExternalVisible := 'False'; ExternalWritable := 'False'} : Bool;   // Transport mode - Run forward request
      sx_SystemReadyRcv { ExternalAccessible := 'False'; ExternalVisible := 'False'; ExternalWritable := 'False'} : Bool;   // System is ready to receive signal
      sx_ParcelInScanningArea { ExternalAccessible := 'False'; ExternalVisible := 'False'; ExternalWritable := 'False'} : Bool;   // Parcel is in scanning area
   END_VAR

   VAR_TEMP
      ti_ScanningWindow : Int;   // Loop counter - To check if some parcel is in the scanning area
   END_VAR


BEGIN
	(*
	----------------------------------------------------------------------------------------
	|                                                                                      |
	|  Copyright  2023             FORTNA Europe BV                                        |
	|  All Rights Reserved         Netherlands                                             |
	|                                                                                      |
	----------------------------------------------------------------------------------------
	Version history:
	Date        | Version   | Author       | Remark
	----------------------------------------------------------------------------------------
	07/03/2023  | 1.0       | S. Nikodem   | Release TIA 17 | DHL Munich 2023
	13/03/2024  | 1.1       | S. Nieswiec  | Added to new baseline
	02/05/2024  | 1.2       | J.Majer      | Datatype conversions changed from automatic to explicit, to accomodate IEC 61131-3 standard
	*)

	REGION 1 - Triggers

	    //Transport mode
	    #R_TRIG_TransportMode(CLK := #sx_TransportmodeOn);

	    //Xray Bag Scaning
	    #R_TRIG_XrayBagScaning(CLK := #ix_XrayBagScaning);
	    #F_TRIG_XrayBagScaning(CLK := #ix_XrayBagScaning);

	    //System is ready to receive
	    //Rising edge trigger
	    #R_TRIG_SystemReadyRcv(CLK := #sx_SystemReadyRcv);
	    //Falling edge trigger
	    #F_TRIG_SystemReadyRcv(CLK := #sx_SystemReadyRcv);

	    //Conveyor runs reverse direction
	    #F_TRIG_ConveyorRunRvs(CLK := #ix_XrayConveyorRunRvs);

	END_REGION

	REGION 2 - Operation conditions
	    //Add doors sensors to conditions

	    #sx_Ready := #ix_SafetyOk
	    AND #ix_24vOk
	    AND #ix_400vOk
	    AND #ix_HardwareOk
	    AND #ix_XrayEnergised
	    AND NOT #ix_XrayFault;

	END_REGION

	REGION 3 - Communication with Xray

	    //When BagScanning signal is active then check at the decision point what parcel is there
	    IF #R_TRIG_XrayBagScaning.Q THEN

	        #iq_UDT_XrayInterface.Communication.SendMessage.GIN := #si_GIN := #iqs_XrayConveyorTrackingData[UDINT_TO_INT(#i_UDT_XrayConfiguration.BagIDPoint)];

	    END_IF;

	    #s_BagScaningTime(iudi_OnDelayTime := #i_UDT_XrayConfiguration.IDmessageTimeout,
	                      ix_SignalToDelay := #ix_XrayBagScaning);

	    IF #s_BagScaningTime.qx_DelayedSignal
	        AND (#si_GIN > 0)
	        AND NOT "DB_GIN".GIN[#si_GIN].DHL.Xray.BagIDMessage.NotReceived
	    THEN

	        //Set variable
	        "DB_GIN".GIN[#si_GIN].DHL.Xray.BagIDMessage.NotReceived := TRUE;

	        //Only for statisctics
	        #ss_Counter.BagIDMessageNotReceived += 1;

	    END_IF;

	    IF #F_TRIG_XrayBagScaning.Q
	        AND NOT "DB_GIN".GIN[#si_GIN].DHL.Xray.BagIDMessage.NotReceived
	    THEN
	        //Set varaible
	        "DB_GIN".GIN[#si_GIN].DHL.Xray.BagIDMessage.Received := True;
	        //Save time
	        "DB_GIN".GIN[#si_GIN].DHL.Xray.BagIDMessage.TimeReceived := #is_ActualTime;

	    END_IF;

	    //Copy send message tirgger to Xray Interface
	    #iq_UDT_XrayInterface.Communication.SendMessage.SendTrigger := #R_TRIG_XrayBagScaning.Q;

	END_REGION

	REGION 4 - Automatic/scan mode

	    //Automatic mode start
	    IF #iq_UDT_EquipmentControl.Command.Start                                                                       // If Start command from from system received
	    THEN
	        #sx_StartReceived := True;

	    END_IF;

	    IF #sx_StartReceived AND
	        #iq_UDT_Handshake.CascadeStartUp
	    THEN

	        #sx_AutomaticOn := TRUE;                                                                            // Set Automatic active
	        #sx_StartReceived := FALSE;                                                                                 // and reset start received bit
	    END_IF;

	    //Automatic mode stop
	    IF (NOT #iq_UDT_EquipmentControl.Command.AutomaticOn                                                             // if Stop active from system control ( Means Not automatic ON)
	        AND NOT #iq_UDT_EquipmentControl.Command.Start                                                              // And no start command from system control
	        AND #sx_AutomaticOn)
	        OR #s_UDT_CommonStatus.Error
	    THEN

	        #sx_AutomaticOn := FALSE;

	    END_IF;

	    //Conveyor before Xray device
	    // Input conveyor is ready to pass a bag to the Xray machine
	    #qx_BHS_RDY_SEND := #sx_AutomaticOn AND #iq_UDT_Handshake.TIP;

	    //Conveyor after Xray device
	    //Output conveyor is ready to accept a bag from the Xray machine
	    #sx_SystemReadyRcv := #sx_AutomaticOn
	    AND #sx_Ready
	    AND #ix_XrayReadyReceive
	    AND #iq_UDT_HandShakeUp.RTR
	    AND (NOT #iq_UDT_XrayInterface.Backbelt.Enable
	    OR (#iq_UDT_XrayInterface.Backbelt.Enable));

	    //Copy static variable to output
	    #qx_BHS_RDY_RCV := #sx_SystemReadyRcv;

	END_REGION

	REGION 5 - Transport mode
	    //Transport mode in automatic mode add condition-     #iq_UDT_OutputConveyor.RTR

	    //Set Transport mode
	    IF #iq_UDT_MFCCommand.TransportModeOn THEN

	        //Set static variable
	        #sx_TransportmodeOn := TRUE;

	        //Reset command
	        #iq_UDT_MFCCommand.TransportModeOn := FALSE;

	        //Only for statisctics
	        #ss_Counter.TransportmodeOn += 1;

	    END_IF;

	    //Reset Transport mode
	    IF #iq_UDT_MFCCommand.TransportModeOff THEN

	        //Set static variable
	        #sx_TransportmodeOn := FALSE;

	        //Reset command
	        #iq_UDT_MFCCommand.TransportModeOff := FALSE;

	        //Only for statisctics
	        #ss_Counter.TransportmodeOff += 1;

	    END_IF;

	    //Copy value to output
	    #qx_TRANSPORT_ENABLE := #sx_TransportmodeOn
	    AND #sx_Ready
	    AND #sx_AutomaticOn;

	    //Run forward request
	    #sx_TransportRunFwd := #sx_TransportmodeOn AND #iq_UDT_HandShakeUp.RTR;

	    #qx_TRANSPORT_FWD := #sx_TransportRunFwd;

	    //Run reverse request - not used
	    #qx_TRANSPORT_REV := FALSE;

	END_REGION

	REGION 6 - Dieback / Backbelt operation

	    REGION 6.1 - Parcel is in the scanning area

	        //Reset varaible
	        #sx_ParcelInScanningArea := False;

	        //Check if some parcel is in the scanning area
	        IF #F_TRIG_SystemReadyRcv.Q THEN

	            FOR #ti_ScanningWindow := #i_UDT_XrayConfiguration.ScanningWindowStartPoint TO #i_UDT_XrayConfiguration.ScanningWindowEndPoint DO

	                IF #iqs_XrayConveyorTrackingData[#ti_ScanningWindow] > 0 THEN

	                    #sx_ParcelInScanningArea := TRUE;

	                END_IF;

	            END_FOR;

	        END_IF;

	    END_REGION

	    REGION 6.2 - Backbelt

	        //Set variable Backbelt if the conditions pass
	        IF #F_TRIG_SystemReadyRcv.Q
	            AND #sx_ParcelInScanningArea
	            AND NOT #ix_XrayReadyReceive
	            AND NOT #ix_XrayConveyorRunFwd
	            AND #iq_UDT_XrayInterface.Backbelt.Enable
	            AND NOT #iq_UDT_XrayInterface.Backbelt.Active
	        THEN

	            #iq_UDT_XrayInterface.Backbelt.Active := True;

	            //Only for staristics
	            #ss_Counter.BackBelt += 1;

	        END_IF;

	        IF (#F_TRIG_ConveyorRunRvs.Q
	            OR #R_TRIG_SystemReadyRcv.Q)
	            AND #iq_UDT_XrayInterface.Backbelt.Active
	        THEN

	            #iq_UDT_XrayInterface.Backbelt.Active := False;

	        END_IF;

	    END_REGION

	END_REGION

	REGION 6 - Handshake

	    //Machine is ready to receive a bag for scanning
	    #iq_UDT_Handshake.RTR := (NOT #sx_TransportmodeOn AND #ix_XrayReadyReceive) OR (#sx_TransportmodeOn AND #ix_XrayConveyorRunFwd);

	    //Machine ready to send a bag from "Exit Sensor"
	    #iq_UDT_HandShakeUp.RTS := (NOT #sx_TransportmodeOn AND #ix_XrayReadySend) OR (#sx_TransportmodeOn AND #ix_XrayConveyorRunFwd);

	END_REGION

	REGION 7 - Errors

	    //Safety reset
	    //Generate pulse
	    #s_EstopReset(iudi_OffDelayTime := #i_UDT_XrayConfiguration.EstopResetPluse,
	                  ix_SignalToDelay := #ix_SafetyReset AND #ix_SafetyOk);

	    #qx_EMERGENCY_STOP_RESET := #s_EstopReset.ix_SignalToDelay;

	    //Estop / To check
	    #qx_ESTOP_IN := #ix_SafetyOk;

	END_REGION


	REGION 8 - Status



	    // Safety not ok
	    #s_UDT_CommonStatus.SafetyStop := NOT #ix_SafetyOk AND #ix_HardwareOk;

	    //Error
	    #s_UDT_CommonStatus.Error := NOT #sx_Ready;

	    // HMI status update
	    IF #s_UDT_CommonStatusOld <> #s_UDT_CommonStatus                                      // update on change

	    THEN
	        // HMI status initialization
	        #s_UDT_HMIStatus.Status := 0;


	        // Safety stop
	        IF (#s_UDT_CommonStatus.SafetyStop)
	        THEN
	            #s_UDT_HMIStatus.Status := "DB_HMIStatusConfiguration".SafetyStop;
	        END_IF;

	        // Error
	        IF (#s_UDT_CommonStatus.Error)
	        THEN
	            #s_UDT_HMIStatus.Status := "DB_HMIStatusConfiguration".Error;
	        END_IF;

	        #s_UDT_CommonStatusOld := #s_UDT_CommonStatus;              // Copy status to memory


	    END_IF;


	    /////////////////////////////////////////////////////////////////////////////////////////////////////////////////////////////////////////

	    // Xray machine errors and arnings
	    #s_UDT_HMIStatus.XraySpecific.XrayEnergised := #ix_XrayEnergised;
	    #s_UDT_HMIStatus.XraySpecific.XrayFault := #ix_XrayFault;
	    #s_UDT_HMIStatus.XraySpecific.XrayRdyRCV := #ix_XrayReadyReceive;
	    #s_UDT_HMIStatus.XraySpecific.XrayRdySend := #ix_XrayReadySend;
	    #s_UDT_HMIStatus.XraySpecific.BagScanning := #ix_XrayBagScaning;
	    #s_UDT_HMIStatus.ConvSpecific.ConvRunFWD := #ix_XrayConveyorRunFwd;
	    #s_UDT_HMIStatus.ConvSpecific.ConvRunREV := #ix_XrayConveyorRunRvs;

	    //Copy value to interface
	    #iq_UDT_XrayInterface.XrayConveyor.RunFwd := #ix_XrayConveyorRunFwd;
	    #iq_UDT_XrayInterface.XrayConveyor.RunRvs := #ix_XrayConveyorRunRvs;

	    //Xray
	    "FC_EquipmentReport"(iUDT_Status := #s_UDT_CommonStatus,
	                         iqUDT_Control := #iq_UDT_EquipmentControl);

	    // Copy HMI status to output
	    #q_UDT_HMIStatus := #s_UDT_HMIStatus;

	END_REGION

	REGION 9 - Statistics

	    // Transport mode active
	    IF (NOT #s_UDT_CommonStatus.Stopped AND #sx_TransportmodeOn)
	        OR #iq_UDT_EquipmentControl.Command.ResetData
	    THEN
	        "FC_Statistics"(ix_Reset := #iq_UDT_EquipmentControl.Command.ResetData,
	                        ix_Activate := NOT #s_UDT_CommonStatus.Stopped AND #sx_TransportmodeOn,
	                        ix_RTrigActivate := #R_TRIG_TransportMode.Q,
	                        iqUDT_Statistics := #iq_UDT_Statistics.TransportMode);
	    END_IF;






	END_REGION

END_FUNCTION_BLOCK

FUNCTION_BLOCK "FB_CodingBeltModes_Van_Line"
{ S7_Optimized_Access := 'TRUE' }
VERSION : 0.1
// ATTRIBUTES
// AUTO_NUMBER = True
// BLOCK_NUMBER = 91
// END_ATTRIBUTES
   VAR_INPUT
      i_UDT_Configuration { ExternalAccessible := 'False'; ExternalVisible := 'False'; ExternalWritable := 'False'} : "UDT_CodingBeltModesConfiguration";   // Function configuration
      ii_Displacement { ExternalAccessible := 'False'; ExternalVisible := 'False'; ExternalWritable := 'False'} : Int;   // Conveyor displacement in one PLC cycle [cm]
      ix_KneeButton { ExternalAccessible := 'False'; ExternalVisible := 'False'; ExternalWritable := 'False'} : Bool;   // Knee button
      ix_LabellingMode { ExternalAccessible := 'False'; ExternalVisible := 'False'; ExternalWritable := 'False'} : Bool;   // Local switch Labeling mode
      ix_ContinueMode { ExternalAccessible := 'False'; ExternalVisible := 'False'; ExternalWritable := 'False'} : Bool;   // Local switch Continue mode
      ix_BufferMode { ExternalAccessible := 'False'; ExternalVisible := 'False'; ExternalWritable := 'False'} : Bool;   // Local switch Buffer mode
      ix_LineModeInfeed { ExternalAccessible := 'False'; ExternalVisible := 'False'; ExternalWritable := 'False'} : Bool;   // Interface with main line - bool or new UDT??? Infeed and Outfeed?
      ix_LineModeOutfeed { ExternalAccessible := 'False'; ExternalVisible := 'False'; ExternalWritable := 'False'} : Bool;   // Interface with main line - bool or new UDT??? Infeed and Outfeed?
      ix_PEC_BoS { ExternalAccessible := 'False'; ExternalVisible := 'False'; ExternalWritable := 'False'} : Bool;   // BoS sensor
      ix_PEC_EoS { ExternalAccessible := 'False'; ExternalVisible := 'False'; ExternalWritable := 'False'} : Bool;   // EoS sensor
   END_VAR

   VAR_OUTPUT
      q_UDT_HMIStatus { ExternalAccessible := 'False'; ExternalVisible := 'False'; ExternalWritable := 'False'} : "UDT_CodingBeltModesStatus";   // Status
      qx_RequestHold_Conveyor { ExternalAccessible := 'False'; ExternalVisible := 'False'; ExternalWritable := 'False'} : Bool;   // Request hold for conveyor
   END_VAR

   VAR
      R_TRIG_KneeButton {InstructionName := 'R_TRIG'; LibVersion := '1.0'; ExternalAccessible := 'False'; ExternalVisible := 'False'; ExternalWritable := 'False'; S7_SetPoint := 'False'} : R_TRIG;   // Rising edge trigger of toogle button
      R_TRIG_LabellingMode {InstructionName := 'R_TRIG'; LibVersion := '1.0'; ExternalAccessible := 'False'; ExternalVisible := 'False'; ExternalWritable := 'False'; S7_SetPoint := 'False'} : R_TRIG;   // Rising edge trigger of labelling mode
      R_TRIG_ContinueMode {InstructionName := 'R_TRIG'; LibVersion := '1.0'; ExternalAccessible := 'False'; ExternalVisible := 'False'; ExternalWritable := 'False'; S7_SetPoint := 'False'} : R_TRIG;   // Rising edge trigger of continue mode
      R_TRIG_BufferMode {InstructionName := 'R_TRIG'; LibVersion := '1.0'; ExternalAccessible := 'False'; ExternalVisible := 'False'; ExternalWritable := 'False'; S7_SetPoint := 'False'} : R_TRIG;   // Rising edge trigger of buffer mode
      R_TRIG_LineModeInfeed {InstructionName := 'R_TRIG'; LibVersion := '1.0'; ExternalAccessible := 'False'; ExternalVisible := 'False'; ExternalWritable := 'False'; S7_SetPoint := 'False'} : R_TRIG;   // Rising edge trigger of Infeed mode
      R_TRIG_LineModeOutfeed {InstructionName := 'R_TRIG'; LibVersion := '1.0'; ExternalAccessible := 'False'; ExternalVisible := 'False'; ExternalWritable := 'False'; S7_SetPoint := 'False'} : R_TRIG;   // Rising edge trigger of Outfeed mode
      R_TRIG_PEC_BoS {InstructionName := 'R_TRIG'; LibVersion := '1.0'; ExternalAccessible := 'False'; ExternalVisible := 'False'; ExternalWritable := 'False'; S7_SetPoint := 'False'} : R_TRIG;   // Falling edge trigger of sensor
      R_TRIG_PEC_EoS {InstructionName := 'R_TRIG'; LibVersion := '1.0'; ExternalAccessible := 'False'; ExternalVisible := 'False'; ExternalWritable := 'False'; S7_SetPoint := 'False'} : R_TRIG;
      sx_LabellingMode { ExternalAccessible := 'False'; ExternalVisible := 'False'; ExternalWritable := 'False'} : Bool;   // Labelling Mode
      sx_ContinueMode { ExternalAccessible := 'False'; ExternalVisible := 'False'; ExternalWritable := 'False'} : Bool;   // Continue Mode
      sx_BufferMode { ExternalAccessible := 'False'; ExternalVisible := 'False'; ExternalWritable := 'False'} : Bool;   // Buffer Mode
      sx_RequestHold { ExternalAccessible := 'False'; ExternalVisible := 'False'; ExternalWritable := 'False'} : Bool;   // Request hold for conveyor
      sx_GeneralError { ExternalAccessible := 'False'; ExternalVisible := 'False'; ExternalWritable := 'False'} : Bool;   // General error
      sx_ConfigurationError { ExternalAccessible := 'False'; ExternalVisible := 'False'; ExternalWritable := 'False'} : Bool;   // Configuration error
      sx_CountDistance { ExternalAccessible := 'False'; ExternalVisible := 'False'; ExternalWritable := 'False'} : Bool;   // Start counting distance to stop position
      sx_ParcelAtPosition { ExternalAccessible := 'False'; ExternalVisible := 'False'; ExternalWritable := 'False'} : Bool;   // The parcel has reached the position
      si_DistanceToStopPosition { ExternalAccessible := 'False'; ExternalVisible := 'False'; ExternalWritable := 'False'} : Int;   // Distance to stop position
   END_VAR


BEGIN
	(*
	----------------------------------------------------------------------------------------
	|                                                                                      |
	|  Copyright  2023             Fortna Europe BV                                        |
	|  All Rights Reserved         Netherlands                                             |
	|                                                                                      |
	|                                                                                      |
	----------------------------------------------------------------------------------------

	Version history:
	Date        | Version   | Author       | Remark
	----------------------------------------------------------------------------------------
	27/07/2023  | 1.0       | S. Nikodem   | Release TIA 17 | DHL Munich 2023
	27/09/2023  | 1.1       | M. Diebel    | Logic changed for two two-position buttons | DHL Munich 2023
	07/02/2024  | 1.2       | L.Klar       | Counting distance fromt he end of the parcel
	12/03/2024  | 1.3       | S. Nieswiec      | Added to new Baseline
	*)

	REGION 1 - Triggers

	    //Knee button
	    #R_TRIG_KneeButton(CLK := (#ix_KneeButton));

	    //Detect end of the parcel
	    //BoS
	    #R_TRIG_PEC_BoS(CLK := #ix_PEC_BoS);
	    //EoS
	    #R_TRIG_PEC_EoS(CLK := #ix_PEC_EoS);

	END_REGION

	REGION 2 - Error detection

	    // Only one mode can be active
	    IF (#ix_LabellingMode AND #ix_ContinueMode)
	        OR (#ix_LabellingMode AND #ix_BufferMode)
	        OR (#ix_ContinueMode AND #ix_BufferMode)
	    THEN

	        #sx_GeneralError := TRUE;

	    ELSE

	        #sx_GeneralError := False;

	    END_IF;

	    //Configuration Error
	    IF #i_UDT_Configuration.LabellingMode_ParcelStop <= 0 THEN

	        #sx_ConfigurationError := TRUE;

	    ELSE

	        #sx_ConfigurationError := False;

	    END_IF;

	END_REGION

	REGION 3 - Modes

	    // Select mode - when the local switch is used or the main line mode is changed

	    #R_TRIG_LabellingMode(CLK := #ix_LabellingMode AND NOT #sx_BufferMode);

	    #R_TRIG_ContinueMode(CLK := (NOT #ix_LabellingMode AND
	                         ((#i_UDT_Configuration.Infeed.LabellingMode AND #ix_LineModeInfeed)
	                         OR (#i_UDT_Configuration.Outfeed.LabellingMode AND #ix_LineModeOutfeed))
	                         OR
	                         NOT #ix_BufferMode AND
	                         ((#i_UDT_Configuration.Infeed.BufferMode AND #ix_LineModeInfeed)
	                         OR (#i_UDT_Configuration.Outfeed.BufferMode AND #ix_LineModeOutfeed))
	                         )
	                         AND
	                         ((#i_UDT_Configuration.Infeed.ContinueMode AND #ix_LineModeInfeed)
	                         OR (#i_UDT_Configuration.Outfeed.ContinueMode AND #ix_LineModeOutfeed)));

	    #R_TRIG_BufferMode(CLK := #ix_BufferMode AND NOT #sx_LabellingMode);

	    #R_TRIG_LineModeInfeed(CLK := #ix_LineModeInfeed);

	    #R_TRIG_LineModeOutfeed(CLK := #ix_LineModeOutfeed);

	    IF #R_TRIG_LabellingMode.Q
	        OR #R_TRIG_ContinueMode.Q
	        OR #R_TRIG_BufferMode.Q
	        OR #R_TRIG_LineModeInfeed.Q
	        OR #R_TRIG_LineModeOutfeed.Q
	    THEN

	        //Clean value from variable when new mode is selected.
	        #sx_LabellingMode := FALSE;
	        #sx_ContinueMode := FALSE;
	        #sx_BufferMode := FALSE;

	        #sx_CountDistance := FALSE;
	        #si_DistanceToStopPosition := 0;
	        #sx_ParcelAtPosition := FALSE;
	        #sx_RequestHold := FALSE;

	        //
	        IF #ix_LabellingMode AND
	            ((#i_UDT_Configuration.Infeed.LabellingMode AND #ix_LineModeInfeed)
	            OR (#i_UDT_Configuration.Outfeed.LabellingMode AND #ix_LineModeOutfeed))
	        THEN

	            #sx_LabellingMode := True;

	        ELSIF
	            (NOT #ix_LabellingMode AND
	            ((#i_UDT_Configuration.Infeed.LabellingMode AND #ix_LineModeInfeed)
	            OR (#i_UDT_Configuration.Outfeed.LabellingMode AND #ix_LineModeOutfeed))
	            OR
	            NOT #ix_BufferMode AND
	            ((#i_UDT_Configuration.Infeed.BufferMode AND #ix_LineModeInfeed)
	            OR (#i_UDT_Configuration.Outfeed.BufferMode AND #ix_LineModeOutfeed))
	            )
	            AND
	            ((#i_UDT_Configuration.Infeed.ContinueMode AND #ix_LineModeInfeed)
	            OR (#i_UDT_Configuration.Outfeed.ContinueMode AND #ix_LineModeOutfeed))
	        THEN

	            #sx_ContinueMode := True;

	        ELSIF
	            #ix_BufferMode AND
	            ((#i_UDT_Configuration.Infeed.BufferMode AND #ix_LineModeInfeed)
	            OR (#i_UDT_Configuration.Outfeed.BufferMode AND #ix_LineModeOutfeed))
	        THEN

	            #sx_BufferMode := True;

	        END_IF;

	    END_IF;

	    REGION 3.1 - Labelling mode

	        IF #sx_LabellingMode THEN

	            IF (#R_TRIG_PEC_BoS.Q AND #ix_LineModeInfeed) OR (#R_TRIG_PEC_EoS.Q AND #ix_LineModeOutfeed) THEN

	                #sx_CountDistance := TRUE;

	            END_IF;

	            //Count the distance to stop parcel position
	            IF #sx_CountDistance THEN

	                #si_DistanceToStopPosition += ABS(#ii_Displacement);

	                IF #si_DistanceToStopPosition > #i_UDT_Configuration.LabellingMode_ParcelStop THEN

	                    #sx_CountDistance := FALSE;
	                    #si_DistanceToStopPosition := 0;
	                    #sx_ParcelAtPosition := True;

	                END_IF;

	            END_IF;

	            //When parcel is at position then stop conveyor
	            #sx_RequestHold := #sx_ParcelAtPosition;

	            //Operator confirm the parcel using knee button
	            IF #R_TRIG_KneeButton.Q THEN

	                #sx_ParcelAtPosition := False;

	            END_IF;


	        END_IF;

	    END_REGION

	    REGION 3.2 - Continue mode

	        IF #sx_ContinueMode THEN

	            IF #R_TRIG_KneeButton.Q THEN

	                #sx_RequestHold := NOT #sx_RequestHold;

	            END_IF;

	        END_IF;

	    END_REGION
	END_REGION

	REGION 4 - Status

	    //Selected mode
	    #q_UDT_HMIStatus.Specific.Infeed_LabellingMode := #sx_LabellingMode AND #ix_LineModeInfeed;
	    #q_UDT_HMIStatus.Specific.Infeed_ContinueMode := #sx_ContinueMode AND #ix_LineModeInfeed;
	    #q_UDT_HMIStatus.Specific.Infeed_BufferMode := #sx_BufferMode AND #ix_LineModeInfeed;
	    #q_UDT_HMIStatus.Specific.Outfeed_LabellingMode := #sx_LabellingMode AND #ix_LineModeOutfeed;
	    #q_UDT_HMIStatus.Specific.Outfeed_ContinueMode := #sx_ContinueMode AND #ix_LineModeOutfeed;
	    #q_UDT_HMIStatus.Specific.Outfeed_BufferMode := #sx_BufferMode AND #ix_LineModeOutfeed;

	    IF (#sx_LabellingMode AND #ix_LineModeInfeed) OR (#sx_LabellingMode AND #ix_LineModeOutfeed)
	    THEN

	        #q_UDT_HMIStatus.Status := "DB_HMIStatusConfiguration".LabbelingMode;

	    END_IF;

	    IF (#sx_ContinueMode AND #ix_LineModeInfeed) OR (#sx_ContinueMode AND #ix_LineModeOutfeed)
	    THEN

	        #q_UDT_HMIStatus.Status := "DB_HMIStatusConfiguration".ContinuousMode;

	    END_IF;

	    IF (#sx_BufferMode AND #ix_LineModeInfeed) OR (#sx_BufferMode AND #ix_LineModeOutfeed)
	    THEN

	        #q_UDT_HMIStatus.Status := "DB_HMIStatusConfiguration".BufferMode;

	    END_IF;

	    IF (NOT #sx_BufferMode AND NOT #sx_ContinueMode AND NOT #sx_LabellingMode AND NOT #ix_LineModeInfeed AND NOT #ix_LineModeOutfeed)
	    THEN

	        #q_UDT_HMIStatus.Status := "DB_HMIStatusConfiguration".Stopped;

	    END_IF;
	    //Errors
	    #q_UDT_HMIStatus.Specific.GeneralError := #sx_GeneralError;
	    #q_UDT_HMIStatus.Specific.ConfigurationError := #sx_ConfigurationError;

	END_REGION

	REGION 5 - Write Output

	    #qx_RequestHold_Conveyor := #sx_RequestHold;

	END_REGION


END_FUNCTION_BLOCK

FUNCTION_BLOCK "FB_ColumnLift"
{ S7_Optimized_Access := 'TRUE' }
VERSION : 0.1
// ATTRIBUTES
// AUTO_NUMBER = True
// BLOCK_NUMBER = 92
// END_ATTRIBUTES
   VAR_INPUT
      i_UDT_ColumnLiftConfiguration { ExternalAccessible := 'False'; ExternalVisible := 'False'; ExternalWritable := 'False'} : "UDT_ColumnLift_Configuration";   // Column lift configuration structure
      ix_SafetyOk { ExternalAccessible := 'False'; ExternalVisible := 'False'; ExternalWritable := 'False'} : Bool;   // TRUE when Safety Circuit of the Conveyor is healthy
      ix_ChuteUpSensor { ExternalAccessible := 'False'; ExternalVisible := 'False'; ExternalWritable := 'False'} : Bool;   // TRUE when upper position sensor is covered
      ix_ChuteDownSensor { ExternalAccessible := 'False'; ExternalVisible := 'False'; ExternalWritable := 'False'} : Bool;   // TRUE when lower position sensor is covered
      ix_LiftUpSensor { ExternalAccessible := 'False'; ExternalVisible := 'False'; ExternalWritable := 'False'} : Bool;   // TRUE when lift up sensor is not covered
      ix_LiftDownSensor { ExternalAccessible := 'False'; ExternalVisible := 'False'; ExternalWritable := 'False'} : Bool;   // TRUE when lift down sensor is not covered
      ix_ChuteNotInPosition { ExternalAccessible := 'False'; ExternalVisible := 'False'; ExternalWritable := 'False'} : Bool;   // TRUE when chut sensor is covered
      ix_PEC_EoS { ExternalAccessible := 'False'; ExternalVisible := 'False'; ExternalWritable := 'False'} : Bool := FALSE;   // TRUE when the end of section photoeye in forward direction is not blocked
      ix_SS_Man { ExternalAccessible := 'False'; ExternalVisible := 'False'; ExternalWritable := 'False'} : Bool;   // TRUE when on Local Controll Panel switch [1] Manual; [0] Automatic
      ix_PB_Down { ExternalAccessible := 'False'; ExternalVisible := 'False'; ExternalWritable := 'False'} : Bool;   // TRUE when on Local Control Panel button Down is on
      ix_PB_Up { ExternalAccessible := 'False'; ExternalVisible := 'False'; ExternalWritable := 'False'} : Bool;   // TRUE when on Local Control Panel button Up is on
      ix_PB_Rst { ExternalAccessible := 'False'; ExternalVisible := 'False'; ExternalWritable := 'False'} : Bool;   // TRUE when on Local Control Panel button reset is on
      ii_Mode { ExternalAccessible := 'False'; ExternalVisible := 'False'; ExternalWritable := 'False'} : Int;   // Mode - [1] Infeed [2] Outfeed
      ix_ChangeModeSignal { ExternalAccessible := 'False'; ExternalVisible := 'False'; ExternalWritable := 'False'} : Bool;   // TRUE when change mode command active
      ix_HardwareOk { ExternalAccessible := 'False'; ExternalVisible := 'False'; ExternalWritable := 'False'} : Bool;   // TRUE when hardware is Ok
      ix_RIONotOnline { ExternalAccessible := 'False'; ExternalVisible := 'False'; ExternalWritable := 'False'} : Bool;
      ix_CaljanLowerOngoing { ExternalAccessible := 'False'; ExternalVisible := 'False'; ExternalWritable := 'False'} : Bool;   // TRUE when the "lower belt" hydraulic valve is active
      ix_CaljanRaisingOngoing { ExternalAccessible := 'False'; ExternalVisible := 'False'; ExternalWritable := 'False'} : Bool;   // TRUE when the "raise belt" hydraulic valve is active
   END_VAR

   VAR_OUTPUT
      q_UDT_HMIStatus { ExternalAccessible := 'False'; ExternalVisible := 'False'; ExternalWritable := 'False'} : "UDT_ColumnLift_Status";   // HMI status structure
      q_UDT_Status { ExternalAccessible := 'False'; ExternalVisible := 'False'; ExternalWritable := 'False'} : "UDT_CommonStatus";   // Common status structure
      qx_ExternalHold { ExternalAccessible := 'False'; ExternalVisible := 'False'; ExternalWritable := 'False'} : Bool;   // External hold for base conveyor
   END_VAR

   VAR_IN_OUT
      iq_UDT_EquipmentControl : "UDT_EquipmentControl";   // Equipment control structure
      iq_UDT_LiftInterface : "UDT_ConveyorInterface";   // Column lift interface
      iq_UDT_Statistics : "UDT_ColumnLift_Statistics";   // Statistics structure
      iq_UDT_HMICommand : "UDT_ColumnLiftCommand";   // Colum lift command from HMI
   END_VAR

   VAR
      s_UDT_HMIStatus { ExternalAccessible := 'False'; ExternalVisible := 'False'; ExternalWritable := 'False'; S7_SetPoint := 'False'} : "UDT_ColumnLift_Status";   // HMI status structure
      s_UDT_StatusOld { ExternalAccessible := 'False'; ExternalVisible := 'False'; ExternalWritable := 'False'; S7_SetPoint := 'False'} : "UDT_CommonStatus";   // Common status structure
      s_UDT_Status { ExternalAccessible := 'False'; ExternalVisible := 'False'; ExternalWritable := 'False'; S7_SetPoint := 'False'} : "UDT_CommonStatus";   // Common status structure
      Jog_Enable { ExternalAccessible := 'False'; ExternalVisible := 'False'; ExternalWritable := 'False'; S7_SetPoint := 'False'} : "FB_TimerOnOffDelay";   // Filtering lower jam photo eye signal
      SwitchingTime { ExternalAccessible := 'False'; ExternalVisible := 'False'; ExternalWritable := 'False'; S7_SetPoint := 'False'} : "FB_TimerOnOffDelay";   // Switching time
      s_FB_Timer_ChuteNoInPosFilter { ExternalAccessible := 'False'; ExternalVisible := 'False'; ExternalWritable := 'False'; S7_SetPoint := 'False'} : "FB_TimerOnOffDelay";   // Chute not in position filter
      s_FB_Timer_LiftUpFilter { ExternalAccessible := 'False'; ExternalVisible := 'False'; ExternalWritable := 'False'; S7_SetPoint := 'False'} : "FB_TimerOnOffDelay";
      R_TRIG_ManualMode {InstructionName := 'R_TRIG'; LibVersion := '1.0'; ExternalAccessible := 'False'; ExternalVisible := 'False'; ExternalWritable := 'False'; S7_SetPoint := 'False'} : R_TRIG;   // Rising edge trigger manual mode
      R_TRIG_ManualJogUp {InstructionName := 'R_TRIG'; LibVersion := '1.0'; ExternalAccessible := 'False'; ExternalVisible := 'False'; ExternalWritable := 'False'; S7_SetPoint := 'False'} : R_TRIG;   // Rising edge trigger manual jog mode command
      R_TRIG_ManualJogDown {InstructionName := 'R_TRIG'; LibVersion := '1.0'; ExternalAccessible := 'False'; ExternalVisible := 'False'; ExternalWritable := 'False'; S7_SetPoint := 'False'} : R_TRIG;   // Rising edge trigger manual jog mode command
      R_TRIG_DownTime {InstructionName := 'R_TRIG'; LibVersion := '1.0'; ExternalAccessible := 'False'; ExternalVisible := 'False'; ExternalWritable := 'False'; S7_SetPoint := 'False'} : R_TRIG;   // Rising edge trigger Column lift is stopped
      R_TRIG_Error {InstructionName := 'R_TRIG'; LibVersion := '1.0'; ExternalAccessible := 'False'; ExternalVisible := 'False'; ExternalWritable := 'False'; S7_SetPoint := 'False'} : R_TRIG;   // Rising edge trigger for Error
      R_TRIG_UpTime {InstructionName := 'R_TRIG'; LibVersion := '1.0'; ExternalAccessible := 'False'; ExternalVisible := 'False'; ExternalWritable := 'False'; S7_SetPoint := 'False'} : R_TRIG;   // Rising edge trigger Column lift is running automatic
      R_TRIG_RestartFromError {InstructionName := 'R_TRIG'; LibVersion := '1.0'; ExternalAccessible := 'False'; ExternalVisible := 'False'; ExternalWritable := 'False'; S7_SetPoint := 'False'} : R_TRIG;   // Rising edge trigger Restart from error
      R_TRIG_PreStartSemiAutomaticUp {InstructionName := 'R_TRIG'; LibVersion := '1.0'; ExternalAccessible := 'False'; ExternalVisible := 'False'; ExternalWritable := 'False'; S7_SetPoint := 'False'} : R_TRIG;   // Rising edge trigger for Pre start semi automatic up signal
      R_TRIG_PreStartSemiAutomaticDown {InstructionName := 'R_TRIG'; LibVersion := '1.0'; ExternalAccessible := 'False'; ExternalVisible := 'False'; ExternalWritable := 'False'; S7_SetPoint := 'False'} : R_TRIG;   // Rising edge trigger for Pre start semi automatic down signal
      R_TRIG_PECUp {InstructionName := 'R_TRIG'; LibVersion := '1.0'; ExternalAccessible := 'False'; ExternalVisible := 'False'; ExternalWritable := 'False'; S7_SetPoint := 'False'} : R_TRIG;   // Rising edge trigger for PEC up position
      R_TRIG_PECDown {InstructionName := 'R_TRIG'; LibVersion := '1.0'; ExternalAccessible := 'False'; ExternalVisible := 'False'; ExternalWritable := 'False'; S7_SetPoint := 'False'} : R_TRIG;   // Rising edge trigger for PEC down position
      F_TRIG_ChuteNotInPosition {InstructionName := 'F_TRIG'; LibVersion := '1.0'; ExternalAccessible := 'False'; ExternalVisible := 'False'; ExternalWritable := 'False'; S7_SetPoint := 'False'} : F_TRIG;   // Falling edge trigger for chute position sensor
      F_TRIG_PECUp {InstructionName := 'F_TRIG'; LibVersion := '1.0'; ExternalAccessible := 'False'; ExternalVisible := 'False'; ExternalWritable := 'False'; S7_SetPoint := 'False'} : F_TRIG;   // Falling edge trigger for PEC up position
      F_TRIG_PECDown {InstructionName := 'F_TRIG'; LibVersion := '1.0'; ExternalAccessible := 'False'; ExternalVisible := 'False'; ExternalWritable := 'False'; S7_SetPoint := 'False'} : F_TRIG;   // Falling edge trigger for PEC down position
      ss_ColumLiftInterface { ExternalAccessible := 'False'; ExternalVisible := 'False'; ExternalWritable := 'False'} : Struct   // Column lift interface static structure
         Positioning { ExternalAccessible := 'False'; ExternalVisible := 'False'; ExternalWritable := 'False'} : Bool;
         SemiAutomatic { ExternalAccessible := 'False'; ExternalVisible := 'False'; ExternalWritable := 'False'} : Bool;
         Manual { ExternalAccessible := 'False'; ExternalVisible := 'False'; ExternalWritable := 'False'} : Bool;
         RunEnabled { ExternalAccessible := 'False'; ExternalVisible := 'False'; ExternalWritable := 'False'} : Bool;
      END_STRUCT;
      sx_StartReceived { ExternalAccessible := 'False'; ExternalVisible := 'False'; ExternalWritable := 'False'} : Bool;   // Start command received from system
      sx_Ready { ExternalAccessible := 'False'; ExternalVisible := 'False'; ExternalWritable := 'False'} : Bool;   // Conveyor Ready to operate in Automatic mode
      sx_SemiAutomatic { ExternalAccessible := 'False'; ExternalVisible := 'False'; ExternalWritable := 'False'} : Bool;   // Running in semi automatic
      sx_PreStartManual { ExternalAccessible := 'False'; ExternalVisible := 'False'; ExternalWritable := 'False'} : Bool;   // Pre conditions to run conveyor in manual mode
      sx_PreStartSemiAutomaticUp { ExternalAccessible := 'False'; ExternalVisible := 'False'; ExternalWritable := 'False'} : Bool;   // Pre conditions to run conveyor in semi automatic up mode
      sx_PreStartSemiAutomaticDown { ExternalAccessible := 'False'; ExternalVisible := 'False'; ExternalWritable := 'False'} : Bool;   // Pre conditions to run conveyor in semi automatic down  mode
      sx_Stopping { ExternalAccessible := 'False'; ExternalVisible := 'False'; ExternalWritable := 'False'} : Bool;   // Stopping is active, first reach position
      sx_SwitchEnable { ExternalAccessible := 'False'; ExternalVisible := 'False'; ExternalWritable := 'False'} : Bool;   // Switching conditions
      sx_UpRequest { ExternalAccessible := 'False'; ExternalVisible := 'False'; ExternalWritable := 'False'} : Bool;   // Request upper outfeed position for actual parcel
      sx_DownRequest { ExternalAccessible := 'False'; ExternalVisible := 'False'; ExternalWritable := 'False'} : Bool;   // Request lower outfeed position for actual parcel
      sx_CombinedJogUp { ExternalAccessible := 'False'; ExternalVisible := 'False'; ExternalWritable := 'False'} : Bool;   // Combined signal of jogging buttons
      sx_CombinedJogDown { ExternalAccessible := 'False'; ExternalVisible := 'False'; ExternalWritable := 'False'} : Bool;   // Combined signal of jogging buttons
      sx_RestartFromError { ExternalAccessible := 'False'; ExternalVisible := 'False'; ExternalWritable := 'False'} : Bool;   // After an error has occurred the action to be done before resuming normal operation
      sx_Jog { ExternalAccessible := 'False'; ExternalVisible := 'False'; ExternalWritable := 'False'} : Bool;   // Off delayed signal Jogging was activated
      sx_ConfigurationError { ExternalAccessible := 'False'; ExternalVisible := 'False'; ExternalWritable := 'False'} : Bool;   // Commissioning: configuration of parameters is wrong
      sx_JogUp { ExternalAccessible := 'False'; ExternalVisible := 'False'; ExternalWritable := 'False'} : Bool;   // Column lift in manual mode - jog up
      sx_JogDown { ExternalAccessible := 'False'; ExternalVisible := 'False'; ExternalWritable := 'False'} : Bool;   // Column lift in manual mode - jog down
      sx_UpperPositionReached { ExternalAccessible := 'False'; ExternalVisible := 'False'; ExternalWritable := 'False'} : Bool;   // Column lift is in upper position
      sx_LowerPositionReached { ExternalAccessible := 'False'; ExternalVisible := 'False'; ExternalWritable := 'False'} : Bool;   // Column lift is in lower position
      sx_MaintenanceControl { ExternalAccessible := 'False'; ExternalVisible := 'False'; ExternalWritable := 'False'} : Bool;   // When maintenance control is active then in manual mode operaton can move column lift to limit swicht
      sx_LiftUpFiltered { ExternalAccessible := 'False'; ExternalVisible := 'False'; ExternalWritable := 'False'} : Bool := TRUE;
   END_VAR

   VAR_TEMP
      ti_ActiveSensor : Int;   // Active sensor counter
   END_VAR

   VAR CONSTANT
      ci_InfeedMode : Int := 1;   // Infeed mode number
      ci_OutfeedMode : Int := 2;   // Outfeed mode number
   END_VAR


BEGIN
	(*
	----------------------------------------------------------------------------------------
	|                                                                                      |
	|  Copyright  2023             FORTNA Europe BV                                        |
	|  All Rights Reserved         Netherlands                                             |
	|                                                                                      |
	----------------------------------------------------------------------------------------
	Version history:
	Date        | Version   | Author       | Remark
	----------------------------------------------------------------------------------------
	11/07/2023  | 1.0       | S. Nikodem   | Release TIA 17 | DHL Munich 2023
	12/09/2023  | 2.0       | M.Diebel     | Addition of AutoOn and Error status upload, Remove hardwareOK from the condition to set warning status
	12/09/2023  | 2.1       | M.Diebel     | New status PositionChangeOngoing instead of running
	05/12/2023  | 2.2       | S. Nikodem   | Functionality update on site
	16/12/2023  | 2.3       | R. Golonka   | HMI command added, HMI status upgrade
	11/01/2024  | 2.4       | L.Klar       | Chute not in position error logic changed
	15/01/2024  | 2.5       | M.Diebel     | Stop on Lift down sensor not on chute down sensor
	17/01/2024  | 2.6       | M.Diebel     | Added filtr for limit UP sensor
	01/02/2024  | 2.7       | M.Diebel     | Added signal from RIO to mask error
	16/02/2024  | 2.8       | M.Diebel     | Add reset for MaintenaceModeActive status
	01/03/2024  | 2.9       | P.Gryszczyk  | Lower position HMI status changed
	13/03/2024  | 2.91      | S. Nieswiec  | Added to new baseline
	*)

	REGION 1 - Initial

	    REGION 1.1 - Triggers

	        // Detecting rising edge on manual mode Or from Equipment Control
	        #R_TRIG_ManualMode(CLK := #s_UDT_Status.Manual);

	        // Rising edge trigger running
	        #R_TRIG_UpTime(CLK := #sx_SemiAutomatic AND #sx_Ready);

	        // Detecting rising edge VSU stopped
	        #R_TRIG_DownTime(CLK := #sx_SemiAutomatic AND NOT #sx_Ready);

	        // Detecting rising edge on VSU error
	        #R_TRIG_Error(CLK := #s_UDT_Status.Error);

	        // Detecting rising edge on start of the restart from error sequence
	        #R_TRIG_RestartFromError(CLK := #sx_RestartFromError);

	        // Detecting falling edge on chute position sensor
	        #F_TRIG_ChuteNotInPosition(CLK := #ix_ChuteNotInPosition);

	        //Maintenance Control
	        #sx_MaintenanceControl := #iq_UDT_HMICommand.MaintenanceControl;

	    END_REGION

	    REGION 1.2 - Filters

	        // Time to start without start warning while jogging
	        #Jog_Enable(iudi_OffDelayTime := #i_UDT_ColumnLiftConfiguration.JogNoHornTime,
	                    ix_SignalToDelay := #sx_Jog);

	        #s_FB_Timer_ChuteNoInPosFilter(iudi_OnDelayTime := 200,
	                                       ix_SignalToDelay := NOT #ix_ChuteDownSensor AND NOT #ix_ChuteNotInPosition);

	        #s_FB_Timer_LiftUpFilter(iudi_OnDelayTime := 100,
	                                 iudi_OffDelayTime := 100,
	                                 ix_SignalToDelay := NOT #ix_LiftUpSensor,
	                                 qx_DelayedSignal => #sx_LiftUpFiltered);

	    END_REGION

	    REGION 1.3 - Switching conditions

	        #sx_SwitchEnable := NOT #iq_UDT_EquipmentControl.Command.StopRequest
	        AND NOT #iq_UDT_LiftInterface.VFDRunning
	        AND NOT #s_UDT_HMIStatus.Specific.ReferenceError
	        AND NOT #s_UDT_HMIStatus.Specific.LimitSensorLowerPosition
	        AND NOT #s_UDT_HMIStatus.Specific.LimitSensorUpperPosition
	        AND NOT #s_UDT_HMIStatus.Specific.ChuteNotInPosition;

	    END_REGION

	    REGION 1.4 - Positioning

	        #ss_ColumLiftInterface.Positioning := #iq_UDT_LiftInterface.ActualSpeed <> 0
	        AND #sx_SemiAutomatic
	        AND NOT #iq_UDT_LiftInterface.InternalErrorVFD;

	    END_REGION

	END_REGION

	REGION 2 - Errors

	    REGION 2.1 - Reset errors

	        //Global reset
	        IF #iq_UDT_EquipmentControl.Command.Reset
	        THEN

	            #s_UDT_HMIStatus.Specific.MaintenaceModeActive := FALSE;
	            #s_UDT_HMIStatus.Specific.SwitchingTimerError := False;

	        END_IF;

	        //Local reset
	        IF #ix_PB_Rst THEN

	            #s_UDT_HMIStatus.Specific.MaintenaceModeActive := FALSE;
	            #s_UDT_HMIStatus.Specific.SwitchingTimerError := False;
	            #s_UDT_HMIStatus.Specific.LimitSensorLowerPosition := False;
	            #s_UDT_HMIStatus.Specific.LimitSensorUpperPosition := False;
	            #s_UDT_HMIStatus.Specific.ChuteNotInPosition := False;

	        END_IF;

	    END_REGION

	    REGION 2.2 - Set errors

	        //Configuration error
	        #sx_ConfigurationError := #i_UDT_ColumnLiftConfiguration.NominalSpeedSetPoint = 0
	        OR #i_UDT_ColumnLiftConfiguration.ManualModeSpeed = 0;

	        //Switching Time
	        #SwitchingTime(iudi_OnDelayTime := #i_UDT_ColumnLiftConfiguration.SwitchingTime,
	                       iudi_OffDelayTime := 0,
	                       ix_SignalToDelay := #sx_SemiAutomatic AND (NOT #iq_UDT_EquipmentControl.Request.SignalingRequest) AND ((#sx_UpRequest AND (NOT #ix_ChuteUpSensor)) OR (#sx_DownRequest AND (NOT #ix_ChuteDownSensor))));

	        IF #SwitchingTime.qx_DelayedSignal THEN
	            #s_UDT_HMIStatus.Specific.SwitchingTimerError := True;
	        END_IF;

	        // Reference error - set error when more like one position sensor is active
	        #ti_ActiveSensor := 0;

	        IF #ix_ChuteUpSensor THEN
	            #ti_ActiveSensor += 1;
	        END_IF;

	        // IF #ix_ChuteDownSensor THEN
	        //     #ti_ActiveSensor += 1;
	        // END_IF;

	        IF NOT #ix_LiftUpSensor THEN
	            #ti_ActiveSensor += 1;
	        END_IF;

	        IF NOT #ix_LiftDownSensor THEN
	            #ti_ActiveSensor += 1;
	        END_IF;

	        IF #ti_ActiveSensor >= 2 AND NOT #ix_RIONotOnline THEN
	            #s_UDT_HMIStatus.Specific.ReferenceError := True;
	        ELSE
	            #s_UDT_HMIStatus.Specific.ReferenceError := False;
	        END_IF;

	    END_REGION

	    REGION 2.3 - Common Error

	        #s_UDT_Status.Error := NOT #ix_HardwareOk
	        OR #iq_UDT_LiftInterface.InternalErrorVFD
	        OR #sx_ConfigurationError
	        OR #s_UDT_HMIStatus.Specific.LimitSensorLowerPosition
	        OR #s_UDT_HMIStatus.Specific.LimitSensorUpperPosition;

	    END_REGION

	    REGION 2.4 - Chute not in position error

	        //Chute not in position
	        IF #s_FB_Timer_ChuteNoInPosFilter.qx_DelayedSignal AND NOT #ix_RIONotOnline THEN
	            //Activate alarm if chuta position is lost
	            #s_UDT_HMIStatus.Specific.ChuteNotInPosition := True;
	        END_IF;

	    END_REGION

	END_REGION

	REGION 3 - Check conditions to set Equipment ready

	    //Conditions to set bit sx_Ready to operate
	    #sx_Ready := NOT #s_UDT_Status.Error                                              // Error not present
	    AND #ix_SafetyOk;                                                                 // Safety signalling OK

	END_REGION

	REGION 4 - Stop Equipment

	    IF (#ix_SS_Man                                                                  // Manual mode is active
	        AND #sx_SemiAutomatic                                                       // Column lift is in semi-automatic mode
	        OR (NOT #iq_UDT_EquipmentControl.Command.AutomaticOn                        // Column lift stops if the bit AutomaticOn from control block is false
	        AND NOT #ix_SS_Man)                                                         // Manual mode active bit
	        OR (NOT #sx_Ready                                                           // Bit column lift ready to run in automatic mode
	        AND NOT #ix_SS_Man)                                                         // Manual mode active
	        OR #ix_SS_Man                                                               // LCP is not set to automatic
	        OR NOT #ix_SafetyOk)                                                        // Safety is not ok
	    THEN
	        #sx_Stopping := TRUE;                                                       // stopping is activated
	        #sx_SemiAutomatic := FALSE;                                                 // switch of automatic activ
	        #sx_StartReceived := FALSE;                                                 // Start command received from system
	    END_IF;

	    IF (#sx_Stopping                                                                 // stopping is activated
	        AND NOT #ss_ColumLiftInterface.Positioning)                                  // The positioning device is not active positioning
	        OR NOT #sx_Ready                                                             // VSU is not ready to run
	    THEN
	        #sx_Stopping := FALSE;                                                       // stopping is activated
	    END_IF;

	END_REGION

	REGION 5 - Start Semi-automatic mode

	    REGION 5.1 - Start

	        // if start (OS) is received from system, this is memorised until started in cascade
	        IF #iq_UDT_EquipmentControl.Command.Start                                       // Start from system
	            AND #sx_Ready                                                               // Equipment has no errors
	        THEN
	            #sx_StartReceived := TRUE;                                                  // Start command received from system
	        END_IF;

	        IF #sx_StartReceived                                                            // Start command received from system
	            AND NOT #ix_SS_Man                                                         // and the LCP is set to auto
	        THEN
	            #sx_SemiAutomatic := TRUE;                                                  // Automatic activated
	            #sx_StartReceived := FALSE;                                                 // Start command received from system
	        END_IF;

	    END_REGION

	END_REGION

	REGION 6 - Manual mode

	    REGION 6.1 - Jog signals

	        #sx_CombinedJogUp := (#ix_SS_Man                                               // box in manual
	        AND #ix_PB_Up);                                                                // If selected jog in positive direction

	        #sx_CombinedJogDown := (#ix_SS_Man                                             // box in manual
	        AND #ix_PB_Down);                                                              // If selected jog in negative direction

	        // Detecting rising edge on manual jog Up
	        #R_TRIG_ManualJogUp(CLK := #sx_CombinedJogUp);

	        // Detecting rising edge on manual jog Down
	        #R_TRIG_ManualJogDown(CLK := #sx_CombinedJogDown);

	    END_REGION

	    REGION 6.2 - Manual mode: disabled

	        // Manual mode bits inputs can be reset in case of malfunction
	        IF NOT #ix_SS_Man
	        THEN
	            #iq_UDT_EquipmentControl.Command.ManualMode := FALSE;                       // reset manual mode command
	            #sx_Jog := FALSE;
	        END_IF;

	    END_REGION

	    REGION 6.3 - Manual PreStart up or down

	        // Pre start conditions to run in manual mode
	        #sx_PreStartManual := #ix_SS_Man                                            // Manual mode active bit
	        AND #ix_SafetyOk                                                            // Safety healthy bit
	        AND NOT #iq_UDT_LiftInterface.InternalErrorVFD;                             // Profinet comunication or PN_DEvice not ok

	        IF #sx_PreStartManual                                                           // Pre start conditions to run in manual mode
	            AND (#R_TRIG_ManualJogUp.Q                                                  // Trigger to start VSU run in manual jog mode UP
	            OR #R_TRIG_ManualJogDown.Q)                                                 // Trigger to start VSU run in manual jog mode Down
	            AND NOT #Jog_Enable.qx_DelayedSignal
	        THEN
	            #iq_UDT_EquipmentControl.Request.SignalingRequest := TRUE;                  // Request signaling TO control block before lift runs in manual mode
	        END_IF;

	    END_REGION

	    REGION 6.4 - Jog mode Up / Down

	        IF #sx_PreStartManual                                                           // IF in manual jog mode
	            AND (NOT #iq_UDT_EquipmentControl.Request.SignalingRequest                  // Signaling request done
	            OR #Jog_Enable.qx_DelayedSignal)
	            AND #sx_CombinedJogUp                                                       // If selected jog in positive direction
	            AND NOT #sx_CombinedJogDown                                                 // And not selected jog in negative direction
	        THEN

	            #sx_JogUp := TRUE;                                                          // set jog positive
	            #sx_JogDown := FALSE;                                                       // reset jog negative
	            #sx_Jog := true;

